// TwinCAT 3 PLC project GFT_drv_demo
// ProgramVersion: 3.1.4024.12
// libraries:
//   Tc2_EtherCAT, * (Beckhoff Automation GmbH)
//   Tc2_Standard, * (Beckhoff Automation GmbH)
//   Tc2_SUPS, * (Beckhoff Automation GmbH)
//   Tc2_System, * (Beckhoff Automation GmbH)
//   Tc2_Utilities, * (Beckhoff Automation GmbH)
//   Tc3_Module, * (Beckhoff Automation GmbH)
//   VisuDialogs, * (System)
//   VisuSymbols,3.5.10.0,System
// project tree:
//   DUTs/ CSdo_State.TcDUT, Ds402_CW.TcDUT, Ds402_Params.TcDUT, Ds402_States.TcDUT, Ds402_SW.TcDUT, E_ModesOfOperation.TcDUT, E_Notes.TcDUT, E_PosTest.TcDUT, E_SquareWave.TcDUT, E_Tests.TcDUT, Mus_Sounds.TcDUT
//   Function Blocks/ FB_Sequence.TcPOU, Profil_CSP.TcPOU
//   / GlobalTextList.TcGTLO, PlcTask.TcTTO, PlcTask_10ms.TcTTO, Visualization Manager.TcVMO (not stored)
//   GVLs/ Ds402.TcGVL, FurElise.TcGVL, GVL_IO.TcGVL, ServoCtrl.TcGVL
//   Image/ ImagePool.TcIPO (not stored)
//   POUs/ FB_PosTest.TcPOU, FB_SineSeq.TcPOU, FB_SquareWave.TcPOU, FB_GetMasterTs.TcPOU, InitSDO.TcPOU, InitSDO_w.TcPOU, MAIN.TcPOU, Main_10ms.TcPOU, MotorOn.TcPOU, OpenExplorer.TcPOU, Prg_GetClock.TcPOU, Prg_logEvents.TcPOU, Prg_WritePersistentVars.TcPOU, processStatusWord.TcPOU, Sequence.TcPOU, TestTorqueProfile.TcPOU
//   RunLog/ F_RunLogSnValid.TcPOU, FB_RunLogger.TcPOU, GVL_RunLog.TcGVL
//   Screen/ Alarm.TcVIS, Control_Panel.TcVIS, Graph.TcVIS, Overview.TcVIS, Overview_ATP.TcVIS, Servo.TcVIS, Settings.TcVIS, Password.TcVIS
//   VISUs/ Visualization.TcVIS
// real-time tasks:
//   TASK PlcTask: cycle T#1ms, priority 8, ADS port 350
//   TASK VISU_TASK: cycle T#200000us, priority 30, ADS port 351
//   TASK PlcTask_10ms: cycle T#10ms, priority 21, ADS port 352
// I/O:
//   DEVICE Device 3 (EtherCAT) (disabled), AmsNetId 5.53.59.176.4.1
//     Term 2 (EK1100) [EK1100 EtherCAT Coupler (2A E-Bus)]
//       Term 3 (EL1859) [EL1859 8Ch. Dig. Input 24V, 3ms, 8Ch. Dig. Output 24V, 0.5A]
//       Term 4 (EL2798) [EL2798 8Ch. Dig. Output 24V AC/DC, 2A, potential-free]
//       Term 5 (EL9011) [EL9011 End Terminal]
//     Box 1 (DOL Drive) [DOL Drive]
// variable links:
//   GFT-drv-demo/GFT-drv-demo Instance <-> Device 3 (EtherCAT)/Box 1 (DOL Drive)
//     PlcTask Inputs/ServoCtrl.ActualCurrent <-> TxPdo-Position-Velocity-Torque Mapping/Torque actual value
//     PlcTask Inputs/ServoCtrl.Position <-> TxPdo-Velocity Mapping/Position actual value
//     PlcTask Inputs/ServoCtrl.StatusWord <-> TxPdo-Velocity Mapping/Statusword
//     PlcTask Outputs/ServoCtrl.ControlWord <-> RxPdo-Position-Velocity-Torque Mapping/Controlword
//     PlcTask Outputs/ServoCtrl.Max_torque0x6072 <-> RxPdo-Position-Velocity-Torque Mapping/Maximal torque
//     PlcTask Outputs/ServoCtrl.ModeOfOperation <-> RxPdo-Position-Velocity-Torque Mapping/Modes of operation
//     PlcTask Outputs/ServoCtrl.PosTarget <-> RxPdo-Position-Velocity-Torque Mapping/Target position
//     PlcTask Outputs/ServoCtrl.TargetTorque <-> RxPdo-Position-Velocity-Torque Mapping/Target Torque
//     PlcTask Outputs/ServoCtrl.Target_velocity0x60FF <-> RxPdo-Position-Velocity-Torque Mapping/Target velocity
//   GFT-drv-demo/GFT-drv-demo Instance <-> Device 3 (EtherCAT)/Term 2 (EK1100)/Term 3 (EL1859)
//     PlcTask Inputs/GVL_IO.ixEmergancy_Stop <-> Channel 1/GVL_IO.ixEmergancy_Stop
//     PlcTask Inputs/GVL_IO.ixGripperLock_1 <-> Channel 4/GVL_IO.ixGripperLock_1
//     PlcTask Inputs/GVL_IO.ixGripperLock_2 <-> Channel 5/GVL_IO.ixGripperLock_1
//     PlcTask Inputs/GVL_IO.ixGripper_Unlock <-> Channel 3/GVL_IO.ixGripper_Unlock
//     PlcTask Inputs/GVL_IO.ixHome_Position <-> Channel 2/GVL_IO.ixHome_Position
//     PlcTask Outputs/GVL_IO.qxEPO_Active <-> Channel 9/GVL_IO.qxEPO_Active
//     PlcTask Outputs/GVL_IO.qxSTO_toDrive <-> Channel 16/GVL_IO.qxSTO_toDrive
//   GFT-drv-demo/GFT-drv-demo Instance <-> Device 3 (EtherCAT)/Term 2 (EK1100)/Term 4 (EL2798)
//     PlcTask Outputs/GVL_IO.qxActuator_1 <-> Channel 1/GVL_IO.qxActuator_1
//     PlcTask Outputs/GVL_IO.qxActuator_2 <-> Channel 2/GVL_IO.qxActuator_2
//     PlcTask Outputs/GVL_IO.qxBrakeOpen <-> Channel 3/GVL_IO.qxBrakeOpen

CONFIGURATION GFT_drv_demo
    RESOURCE PLC ON TwinCAT3
        TASK PlcTask(INTERVAL := T#1ms, PRIORITY := 8);
        TASK PlcTask_10ms(INTERVAL := T#10ms, PRIORITY := 21);
        PROGRAM MAIN WITH PlcTask : MAIN;
        PROGRAM Main_10ms WITH PlcTask_10ms : Main_10ms;
    END_RESOURCE
END_CONFIGURATION

// ---- DUTs/CSdo_State.TcDUT
TYPE CSdo_State :
STRUCT
	nIndex          : WORD;
	nSubIndex       : BYTE;
	bExecute        : BOOL := TRUE;
	bError			: BOOL;
	nErrId 			: UDINT;
	nBufLen   		: UDINT; 
	pBuf			: PVOID;	
END_STRUCT
END_TYPE

// ---- DUTs/Ds402_CW.TcDUT

TYPE Ds402_CW:
STRUCT 
	ReadyToSwitchOn : BOOL;// = bitand(sw,1);
	SwitchOn : BOOL;//= bitand(bitshift(sw,-1),1);
	OperationEnabled : BOOL;// = bitand(bitshift(sw,-2),1);
	Fault : BOOL;// = bitand(bitshift(sw,-3),1);
	VoltageEnabled : BOOL;// = bitand(bitshift(sw,-4),1);
	NoQuickStop : BOOL;// = bitand(bitshift(sw,-5),1);
	SwitchOnDisabled : BOOL;// = bitand(bitshift(sw,-6),1);
	Warning : BOOL;// = bitand(bitshift(sw,-7),1);
	ManufacturerSpecific8 : BOOL;// = bitand(bitshift(sw,-8),1);
	Remote : BOOL;// = bitand(bitshift(sw,-9),1);
	TargetReached : BOOL;// = bitand(bitshift(sw,-10),1);
	InternalLimitActive : BOOL;// = bitand(bitshift(sw,-11),1);
	OperationModeSpecific12to13 : INT;// = bitand(bitshift(sw,-12),3);
	ManufacturerSpecific14to15 : INT;// = bitand(bitshift(sw,-14),3);
END_STRUCT
END_TYPE

// ---- DUTs/Ds402_Params.TcDUT
TYPE Ds402_Params :
STRUCT
	Motor_rated_torque0x6076 : UDINT;
	Interpolation_time_period0x60C2_1_period : USINT;
	Interpolation_time_period0x60C2_2_period : SINT;
	vendorId_0x1081_1 : UDINT;
	Postion_window0x6067 : UDINT;
	Position_window_time0x6068 :  UINT;
	Abort_connection_option_code_0x6007 :  UINT;
	Torque_slope0x6087 :    UDINT;
END_STRUCT
END_TYPE

// ---- DUTs/Ds402_States.TcDUT
{attribute 'qualified_only'}
{attribute 'strict'}
(*
TYPE Ds402_States :
(
	FSM_Ilegal := -2 ;
	FSM_NotReadyToSwitchOn := -1 ; 
	FSM_SwitchOnDisabled  := 0 ;
	FSM_ReadyToSwitchOn := 1;
	FSM_SwitchedOn := 2;
	FSM_OperationEnabled := 3 ;
	FSM_QuickStopActive := 4 ;
	FSM_FaultReactionActive := 5;
	FSM_Fault := 6 ; 
	FSM_Temporary_Fault := 7; 
);
END_TYPE
*)
;

// ---- DUTs/Ds402_SW.TcDUT
TYPE Ds402_SW :
STRUCT
	ReadyToSwitchOn : BOOL;// = bitand(sw,1);
	SwitchOn : BOOL;//= bitand(bitshift(sw,-1),1);
	OperationEnabled : BOOL;// = bitand(bitshift(sw,-2),1);
	Fault : BOOL;// = bitand(bitshift(sw,-3),1);
	VoltageEnabled : BOOL;// = bitand(bitshift(sw,-4),1);
	NoQuickStop : BOOL;// = bitand(bitshift(sw,-5),1);
	SwitchOnDisabled : BOOL;// = bitand(bitshift(sw,-6),1);
	Warning : BOOL;// = bitand(bitshift(sw,-7),1);
	ManufacturerSpecific8 : BOOL;// = bitand(bitshift(sw,-8),1);
	Remote : BOOL;// = bitand(bitshift(sw,-9),1);
	TargetReached : BOOL;// = bitand(bitshift(sw,-10),1);
	InternalLimitActive : BOOL;// = bitand(bitshift(sw,-11),1);
	OperationModeSpecific12to13 : INT;// = bitand(bitshift(sw,-12),3);
	ManufacturerSpecific14to15 : INT;// = bitand(bitshift(sw,-14),3);

	SetPointAck:   BOOL ;// bitand(bitshift(sw,-12),1);
	FollowingError:BOOL ; // bitand(bitshift(sw,-13),1);

END_STRUCT
END_TYPE

// ---- DUTs/E_ModesOfOperation.TcDUT
{attribute 'qualified_only'}
{attribute 'strict'}
TYPE E_ModesOfOperation :
(
	ED_MO_NoModeChange := 0 , 
	ED_MO_Profile_position_mode := 1 , 
	ED_MO_Profile_velocity_mode := 3 , 
	ED_MO_Torque_profile_mode := 4, 
	ED_MO_Inertial_profile_mode := 5, 
	ED_MO_Homing_mode := 6, 
	ED_MO_Interpolated_position_mode := 7, 
	ED_MO_Cyclic_sync_position_mode := 8, 
	ED_MO_Cyclic_sync_velocity_mode := 9, 
	ED_MO_Cyclic_sync_torque_mode := 10,
	ED_MO_Profile_only_velocity_mode := 11,
	ED_MO_Profile_test_wave_mode := 12,
	ED_MO_User_Prj_spec_mode := 13
);
END_TYPE

// ---- DUTs/E_Notes.TcDUT
{attribute 'qualified_only'}
{attribute 'strict'}
TYPE E_Notes :
(
STOP     := 0,
PAUSE    := 1,
NOTE_B0  := 31  ,
NOTE_C1  := 33  ,
NOTE_CS1 := 35  ,
NOTE_D1  := 37  ,
NOTE_DS1 := 39  ,
NOTE_E1  := 41  ,
NOTE_F1  := 44  ,
NOTE_FS1 := 46  ,
NOTE_G1  := 49  ,
NOTE_GS1 := 52  ,
NOTE_A1  := 55  ,
NOTE_AS1 := 58  ,
NOTE_B1  := 62  ,
NOTE_C2  := 65  ,
NOTE_CS2 := 69  ,
NOTE_D2  := 73  ,
NOTE_DS2 := 78  ,
NOTE_E2  := 82  ,
NOTE_F2  := 87  ,
NOTE_FS2 := 93  ,
NOTE_G2  := 98  ,
NOTE_GS2 := 104 ,
NOTE_A2  := 110 ,
NOTE_AS2 := 117 ,
NOTE_B2  := 123 ,
NOTE_C3  := 131 ,
NOTE_CS3 := 139 ,
NOTE_D3  := 147 ,
NOTE_DS3 := 156 ,
NOTE_E3  := 165 ,
NOTE_F3  := 175 ,
NOTE_FS3 := 185 ,
NOTE_G3  := 196 ,
NOTE_GS3 := 208 ,
NOTE_A3  := 220 ,
NOTE_AS3 := 233 ,
NOTE_B3  := 247 ,
NOTE_C4  := 262 ,
NOTE_CS4 := 277 ,
NOTE_D4  := 294 ,
NOTE_DS4 := 311 ,
NOTE_E4 := 330 ,
NOTE_F4  := 349 ,
NOTE_FS4 := 370 ,
NOTE_G4  := 392 ,
NOTE_GS4 := 415 ,
NOTE_A4  := 440 ,
NOTE_AS4 := 466 ,
NOTE_B4  := 494 ,
NOTE_C5  := 523 ,
NOTE_CS5 := 554 ,
NOTE_D5  := 587 ,
NOTE_DS5 := 622 ,
NOTE_E5  := 659 ,
NOTE_F5  := 698 ,
NOTE_FS5 := 740 ,
NOTE_G5  := 784 ,
NOTE_GS5 := 831 ,
NOTE_A5  := 880 ,
NOTE_AS5 := 932 ,
NOTE_B5  := 988 ,
NOTE_C6  := 1047,
NOTE_CS6 := 1109,
NOTE_D6  := 1175,
NOTE_DS6 := 1245,
NOTE_E6  := 1319,
NOTE_F6  := 1397,
NOTE_FS6 := 1480,
NOTE_G6  := 1568,
NOTE_GS6 := 1661,
NOTE_A6  := 1760,
NOTE_AS6 := 1865,
NOTE_B6  := 1976,
NOTE_C7  := 2093,
NOTE_CS7 := 2217,
NOTE_D7  := 2349,
NOTE_DS7 := 2489,
NOTE_E7  := 2637,
NOTE_F7  := 2794,
NOTE_FS7 := 2960,
NOTE_G7  := 3136,
NOTE_GS7 := 3322,
NOTE_A7  := 3520,
NOTE_AS7 := 3729,
NOTE_B7  := 3951,
NOTE_C8  := 4186,
NOTE_CS8 := 4435,
NOTE_D8  := 4699,
NOTE_DS8 := 4978
);
	
END_TYPE

// ---- DUTs/E_PosTest.TcDUT
{attribute 'qualified_only'}
{attribute 'strict'}
TYPE E_PosTest :
(
	Idle_start :=0,
	GoToNextState_levelHi := 1,
	GoToNextState_levelLo := 2,
	MovingTo_levelHi :=3,
	MovingTo_levelLo :=4,
	Idle_init :=5
);
END_TYPE

// ---- DUTs/E_SquareWave.TcDUT
{attribute 'qualified_only'}
{attribute 'strict'}
TYPE E_SquareWave :
(
	GoToNextState_levelHi := 1,
	GoToNextState_levelLo :=2,
	GoToNextState_Off :=3
);
END_TYPE

// ---- DUTs/E_Tests.TcDUT
{attribute 'qualified_only'}
{attribute 'strict'}
TYPE E_Tests :
(
	E_Current_SquareWaveTest := 1,
	E_Current_SinWaveTest := 2,
	E_Position_Ptp := 3,
	E_Position_Csp := 4,
	E_Velocity_Csv :=5
);
END_TYPE

// ---- DUTs/Mus_Sounds.TcDUT
TYPE Mus_Sounds :
STRUCT
	note : E_Notes;
	tempo: INT;
END_STRUCT
END_TYPE

// ---- GVLs/Ds402.TcGVL
{attribute 'qualified_only'}


VAR_GLOBAL
	StatusWord_Bits :  Ds402_SW;
	DirUp : BOOL;
	ProfParams : Ds402_Params;

END_VAR

// ---- GVLs/FurElise.TcGVL
{attribute 'qualified_only'}
VAR_GLOBAL CONSTANT
	FurElise : ARRAY [0..100] OF  Mus_Sounds :=[
 	(note := E_Notes.NOTE_E5,              tempo:= 9),
                (note := E_Notes.NOTE_DS5,  tempo:=    9),
                (note := E_Notes.NOTE_E5,    tempo:=   9),
                (note := E_Notes.NOTE_DS5,   tempo:=   9),
                (note := E_Notes.NOTE_E5,    tempo:=   9),
                (note := E_Notes.NOTE_B4,    tempo:=   9),
                (note := E_Notes.NOTE_D5,    tempo:=   9),
                (note := E_Notes.NOTE_C5,    tempo:=   9),
                (note := E_Notes.NOTE_A4,    tempo:=   3),
                (note := E_Notes.NOTE_C4,    tempo:=   9),
                (note := E_Notes.NOTE_E4,    tempo:=   9),
                (note := E_Notes.NOTE_A4,    tempo:=   9),
                (note := E_Notes.NOTE_B4,     tempo:=  3),
                (note := E_Notes.NOTE_E4,    tempo:=   9),
                (note := E_Notes.NOTE_GS4,    tempo:=  9),
                (note := E_Notes.NOTE_B4,    tempo:=          9),
                (note := E_Notes.NOTE_C5,    tempo:=   3),
                (note := E_Notes.NOTE_E4,    tempo:=   9),
                (note := E_Notes.NOTE_E5,    tempo:=   9),
                (note := E_Notes.NOTE_DS5,   tempo:=   9),
                (note := E_Notes.NOTE_E5,    tempo:=   9),
                (note := E_Notes.NOTE_DS5,   tempo:=   9),
                (note := E_Notes.NOTE_E5,    tempo:=   9),
                (note := E_Notes.NOTE_B4,    tempo:=   9),
                (note := E_Notes.NOTE_D5,   tempo:=    9),
                (note := E_Notes.NOTE_C5,   tempo:=    9),
                (note := E_Notes.NOTE_A4,    tempo:=   3),
                (note := E_Notes.NOTE_C4,    tempo:=   9),
                (note := E_Notes.NOTE_E4,    tempo:=   9),
                (note := E_Notes.NOTE_A4,    tempo:=   9),
                (note := E_Notes.NOTE_B4,    tempo:=   3),
                (note := E_Notes.NOTE_E4,    tempo:=          9),
                (note := E_Notes.NOTE_C5,    tempo:=   9),
                (note := E_Notes.NOTE_B4,   tempo:=    9),
                (note := E_Notes.NOTE_A4,    tempo:=   3),
                (note := E_Notes.NOTE_B4,    tempo:=   9),
                (note := E_Notes.NOTE_C5,    tempo:=   9),
                (note := E_Notes.NOTE_D5,    tempo:=   9),
                (note := E_Notes.NOTE_E5,    tempo:=   3),
                (note := E_Notes.NOTE_G4,    tempo:=   9),
                (note := E_Notes.NOTE_F5,    tempo:=   9),
                (note := E_Notes.NOTE_E5,    tempo:=   9),
                (note := E_Notes.NOTE_D5,     tempo:=  3),
                (note := E_Notes.NOTE_F4,     tempo:=  9),
                (note := E_Notes.NOTE_E5,    tempo:=   9),
                (note := E_Notes.NOTE_D5,    tempo:=   9),
                (note := E_Notes.NOTE_C5,    tempo:=   3),
                (note := E_Notes.NOTE_E4,    tempo:=          9),
                (note := E_Notes.NOTE_D5,   tempo:=    9),
                (note := E_Notes.NOTE_C5,    tempo:=   9),
                (note := E_Notes.NOTE_B4,    tempo:=   9),
                (note := E_Notes.NOTE_E4,    tempo:=   9),
                (note := E_Notes.NOTE_E5,   tempo:=    9),
                (note := E_Notes.NOTE_E4,    tempo:=   9),
                (note := E_Notes.NOTE_E5,    tempo:=   9),
                (note := E_Notes.NOTE_E4,    tempo:=   9),
                (note := E_Notes.NOTE_E5,    tempo:=   9),
                (note := E_Notes.NOTE_E4,     tempo:=  9),
                (note := E_Notes.NOTE_E5,    tempo:=   9),
                (note := E_Notes.NOTE_DS4,    tempo:=  9),
                (note := E_Notes.NOTE_E5,    tempo:=   9),
                (note := E_Notes.NOTE_D4,     tempo:=  9),
                (note := E_Notes.NOTE_E5,     tempo:=  9),
                (note := E_Notes.NOTE_DS4,   tempo:=        9),
                (note := E_Notes.NOTE_E5,    tempo:=   9),
                (note := E_Notes.NOTE_B4,    tempo:=   9),
                (note := E_Notes.NOTE_D5,    tempo:=   9),
                (note := E_Notes.NOTE_C5,    tempo:=   9),
                (note := E_Notes.NOTE_A4,     tempo:=  3),
                (note := E_Notes.NOTE_C4,     tempo:=  9),
                (note := E_Notes.NOTE_E4,    tempo:=   9),
                (note := E_Notes.NOTE_A4,    tempo:=   9),
                (note := E_Notes.NOTE_B4,    tempo:=   3),
                (note := E_Notes.NOTE_E4,    tempo:=   9),
                (note := E_Notes.NOTE_GS4,   tempo:=   9),
                (note := E_Notes.NOTE_B4,     tempo:=  9),
                (note := E_Notes.NOTE_C5,     tempo:=  3),
                (note := E_Notes.NOTE_E4,     tempo:=  9),
                (note := E_Notes.NOTE_E5,     tempo:=  9),
                (note := E_Notes.NOTE_DS5,    tempo:=       9),
                (note := E_Notes.NOTE_E5,    tempo:=   9),
                (note := E_Notes.NOTE_DS5,    tempo:=  9),
                (note := E_Notes.NOTE_E5,     tempo:=  9),
                (note := E_Notes.NOTE_B4,     tempo:=  9),
                (note := E_Notes.NOTE_D5,     tempo:=  9),
                (note := E_Notes.NOTE_C5,     tempo:=  9),
                (note := E_Notes.NOTE_A4,    tempo:=   3),
                (note := E_Notes.NOTE_C4,    tempo:=   9),
                (note := E_Notes.NOTE_E4,    tempo:=   9),
                (note := E_Notes.NOTE_A4,    tempo:=   9),
                (note := E_Notes.NOTE_B4,    tempo:=   3),
                (note := E_Notes.NOTE_E4,    tempo:=   8),
                (note := E_Notes.NOTE_C5,    tempo:=   8),
                (note := E_Notes.NOTE_B4,    tempo:=   8),
                (note := E_Notes.NOTE_A4,    tempo:=   1),
                (note := E_Notes.STOP,       tempo:=   9)
];

END_VAR

// ---- GVLs/GVL_IO.TcGVL
{attribute 'qualified_only'}
VAR_GLOBAL
	
	// Digital Input
	ixGripper_Up AT%I*:BOOL;
	ixEncoder AT%I*:BOOL;
	ixHome_Position AT%I*:BOOL;
	ixEmergancy_Stop AT%I*:BOOL;
	ixGripperLock_1 AT%I*:BOOL;
	ixGripperLock_2 AT%I*:BOOL;
	ixGripper_Unlock AT%I*:BOOL;
	ixGripperLock_A AT%I*:BOOL;
	ixGripperLock_B AT%I*:BOOL;
	
	
	//MOtor input
	Velosity_PV AT%I*:DINT;
	
	// Digital Output
	qxStart_Motor AT%Q*:BOOL;
	qxOpen_Gripper AT%Q*:BOOL;
	qxGripper_UP AT%Q*:BOOL;
	qxSTO_toDrive AT%Q*:BOOL;
	qxEPO_Active AT%Q*:BOOL;
	qxClose_Gripper AT%Q*:BOOL;
	qxBrakeOpen AT%Q*:BOOL;
	qxActuator_1 AT%Q*:BOOL; 	// Direction : 0 - close; 1 - open
	qxActuator_2 AT%Q*:BOOL;	// command Move 
	
	// Global
	Reset, Homing, Motor_UP, Motor_DN, Gripper_Open_cmd, Gripper_Close_cmd, Jog_UP, Jog_DN , Zeroing_cmd: BOOL;
	Position_PV, Position_SP, Motor_I , Position_PV_HMI, Position_PV_Diff: DINT;
	 
	Motor_I_PV, Motor_I_MAX, Motor_I_AVR : REAL;
	Motor_I_mem : ARRAY [0..500] OF REAL;
	Position_PV_mem : ARRAY [0..500] OF DINT;
	
	
	Enable, Emergancy_OK, Motor_UP_cmd, Motor_DN_cmd, Homing_OK, Homing_cmd , TwoSensorLock:BOOL;
	Step, Gripper_step:INT;
	Always_ON, Always_OFF, FirstScan :BOOL;
	GO_TO_cmd, Motion_in_Progress, Ready_for_start, Start, Stop, Run_Cycle, Enable_motor_cmd:BOOL;
	tonHomingError_IN, tonHomingStepDelay_IN : BOOL;
	tonHomingStepDelay_SP : TIME;
	
	 
	
	
	Position_UP_SP_LL, Position_UP_SP_HL, Position_DN_SP_LL, Position_DN_SP_HL : DINT;
	Cycle_PV: UDINT;
	UP_pause_in:BOOL;
	Error, Gripper_Open_Error, Gripper_Close_Error , Emergancy_Error, SensorLock_Error, Homing_Error, Motor_Error: BOOL;
	Position_sp_test : DINT;
	pp, pv :REAL;
	Speed_SP_mem, Accseleration_SP_mem : REAL;
	tonUserDelay_IN, tonUserDelay_Q, tonMotionError_IN, tonMotionError_Q : BOOL;
	tonLogTimer_IN , tonLogTimer_Q : BOOL;
	Password : INT := 9118 ;
	Password_IN : INT;
	
	Calc_log_cmd , OpenExplorer_cmd, New_CSV_cmd : BOOL;
	Lod_appendLine_cmd, Log_CloseFile_cmd : BOOL;
	Log_nMode : DWORD;
	Log_Data, Motor_UP_slow_cmd, Motor_DN_slow_cmd , Slow_cycle_cmd , ATP_start_cmd: BOOL;	
	test_Gripper_open_OK, test_Gripper_close_OK, test_motor_sldown_ok, test_motor_slUP_ok, test_Insert_OK, test_slowCycle_OK : BOOL;
		
	
	
	
END_VAR

VAR_GLOBAL PERSISTENT
	vcc_SP : REAL ; //:= 4000000;
	acc_SP: REAL ; //:= 80000000;
    Position_UP_SP, Position_DN_SP : DINT;
	Position_UP_A_SP, Position_DN_A_SP : DINT; // position  Accseleration Change
	Speed_SP, Accseleration_SP , Accseleration_A_SP: REAL;
	Speed_SP_slow, Accseleration_SP_slow : REAL;
	Cycle_SP : UDINT;
	Motor_Limit_UP, Motor_Limit_DN :DINT; 
	
	
	
	
END_VAR

// ---- GVLs/ServoCtrl.TcGVL
{attribute 'qualified_only'}
VAR_GLOBAL
	TargetTorque AT %Q*: INT;
	TorqueProfState: REAL;
	PosTarget  AT %Q*: DINT;
	Position  AT %I*: DINT ;
	ControlWord AT %Q*: UINT;
	StatusWord AT %I*:  INT ;
	ActualCurrent AT %I*:  DINT ;
	ModeOfOperation AT %Q*: SINT;
	PosSensor1 AT %I*:  DINT ;
	PosSensor2 AT %I*:  DINT ;
	Max_torque0x6072 AT %Q*: UINT;
	Target_velocity0x60FF AT %Q*: DINT;
END_VAR

// ---- RunLog/GVL_RunLog.TcGVL
// Run log module: what the HMI shows and enters. Format: report-tool/docs/log-format.md
{attribute 'qualified_only'}
VAR_GLOBAL
	SN			: STRING(32);	// part serial number, entered on Overview_ATP before START
	SN_valid	: BOOL;			// 1..32 characters of A-Z a-z 0-9 -; ATP START needs it
	State		: STRING(40);	// what the logger is doing now
	LastFile	: STRING(255);	// last finished run log
	LastError	: STRING(255);	// last problem; a run without a valid SN is not logged
	ErrorCount	: UDINT;
END_VAR

// ---- POUs/MAIN.TcPOU
PROGRAM MAIN
VAR

testType : E_Tests :=E_Tests.E_Position_Csp;// E_Tests.E_Velocity_Csv;//E_Tests.E_Position_Csp;//E_Tests.E_Current_SinWaveTest;//E_Tests.E_Position_Ptp;

ApplyPosTargetNow : BOOL := FALSE;
//ModeOfOperation : SINT := TO_SINT(E_ModesOfOperation.ED_MO_Cyclic_sync_torque_mode);// ED_MO_Cyclic_sync_torque_mode
bInitDone : BOOL :=FALSE;
bInitDone_w : BOOL :=FALSE;//finished SDO download to slave

valueA : UDINT;
sNetId     : T_AmsNetId := '5.53.59.176.4.1'; // '5.53.59.176.1.1';
nSlaveAddr : UINT := 1001;
//fbSdoRead  : FB_EcCoESdoRead;
//sdo1_err : BOOL;
//sdo1_nErrId : UDINT;
//sdo1_value  :  UDINT;
//sdo1_value_size  :  UDINT := SIZEOF(sdo1_value);

TorCmd_ds402  :  INT :=0;
TorCmdMax_Ds402 :  UINT :=0;
TorCmdA : REAL := 4;
TorCmdMaxA : REAL := 17;
FreqScale : REAL := 0.25;
ProfParams: Ds402_Params;// uploaded from slave
ProfParams_w: Ds402_Params;// to download to slave
// State machine
fbSquareWave		: FB_SquareWave;
fbMusic : FB_SineSeq;
fbInitSDO_w : InitSDO_w;// write SDO to slave
fbInitSDO : InitSDO;// read SDO from slave
fbPosTest : FB_PosTest; // position profiler test

	bInit_Sdo_States : BOOL :=TRUE;
//	indSdo :   USINT :=0;
//	Sdo_States : ARRAY [0..10] OF CSdo_State ;
	TaskTotalTime : UDINT;
	fbGetMasterTs : FB_GetMasterTs;
	cpu_info : ARRAY [0..10] of ST_CpuCoreInfo;
	FB_Sequence_DB: FB_Sequence;
	Profile_CSP_DB: Profil_CSP;
	
	
	
	
END_VAR


TaskTotalTime := F_GetTaskTotalTime(0);// x100ns 
fbGetMasterTs();
F_GetCpuCoreInfo(0,ADR(cpu_info[0]));
F_GetCpuCoreInfo(0,ADR(cpu_info[1]));
 
(*
IF bInit_Sdo_States AND fbGetMasterTs.MasterTsUsec> 0 THEN
	fbInitSDO(sNetId:=sNetId,nSlaveAddr:=nSlaveAddr);
	fbInitSDO.Init();

	CASE fbGetMasterTs.MasterTsUsec OF
	100:
		ProfParams_w.Interpolation_time_period0x60C2_1_period := 10;
		ProfParams_w.Interpolation_time_period0x60C2_2_period := -5;
	200:
		ProfParams_w.Interpolation_time_period0x60C2_1_period := 20;
		ProfParams_w.Interpolation_time_period0x60C2_2_period := -5;
		
	250:
		ProfParams_w.Interpolation_time_period0x60C2_1_period := 25;
		ProfParams_w.Interpolation_time_period0x60C2_2_period := -5;
	
	500:
		ProfParams_w.Interpolation_time_period0x60C2_1_period := 5;
		ProfParams_w.Interpolation_time_period0x60C2_2_period := -4;
	1000:
		ProfParams_w.Interpolation_time_period0x60C2_1_period := 1;
		ProfParams_w.Interpolation_time_period0x60C2_2_period := -3;
	END_CASE
	ProfParams_w.Postion_window0x6067 := 200;
	ProfParams_w.Position_window_time0x6068 := 1000;
	
	ProfParams_w.Abort_connection_option_code_0x6007 := 16#0002;
	
	fbInitSDO_w(sNetId:=sNetId,nSlaveAddr:=nSlaveAddr,ProfParams:=ProfParams_w);
	fbInitSDO_w.Init();
	//FreqScale := 0.25 * 1000.0 / INT_TO_REAL(fbGetMasterTs.MasterTsUsec)   ;
	bInit_Sdo_States:= FALSE;
END_IF

IF NOT bInit_Sdo_States THEN
	fbInitSDO_w.writeSDO();
	bInitDone_w := fbInitSDO_w.bInitDone;
	IF bInitDone_w THEN
	fbInitSDO.readSDO();
	bInitDone := fbInitSDO.bInitDone;
	END_IF
END_IF
*)
bInitDone:= TRUE;
//TestTorqueProfile();
IF bInitDone THEN
	ProfParams:= fbInitSDO.ProfParams;
	
	//IF ProfParams.Motor_rated_torque0x6076 > 0 THEN
	//	TorCmd_ds402  := TRUNC_INT( TorCmdA * 1E6 / UDINT_TO_REAL(ProfParams.Motor_rated_torque0x6076));// TC*10e6/0x6076
	//	TorCmdMax_Ds402:=INT_TO_UINT( TRUNC_INT( TorCmdMaxA * 1E6 / UDINT_TO_REAL(ProfParams.Motor_rated_torque0x6076)));// TC*10e6/0x6076
	//ELSE 
	//	TorCmd_ds402  :=0;TorCmdMax_Ds402:=0;
	//END_IF
	TorCmdMax_Ds402:= 65535;//62000;
	
	// E_Current_SquareWaveTest->E_Current_SinWaveTest->E_Position_Ptp
	CASE testType OF
		E_Tests.E_Current_SquareWaveTest:
			fbSquareWave(RefLevelHi:= TorCmd_ds402,RefLevelLo:= -TorCmd_ds402);
			fbSquareWave.Execute(bCyclicMode:=FALSE);
			IF fbSquareWave.nCycles > 20 THEN
				fbSquareWave.Restart();
				testType := E_Tests.E_Current_SinWaveTest;
			END_IF
		E_Tests.E_Current_SinWaveTest:
			fbMusic(Motor_rated_torque0x6076:=ProfParams.Motor_rated_torque0x6076,
			AmpMax := TorCmdMaxA,FreqScale:= FreqScale);
			fbMusic.Execute(Mode_of_operation:= E_ModesOfOperation.ED_MO_Cyclic_sync_torque_mode);
			IF fbMusic.nCycles > 0 THEN
				fbMusic.Restart();
				testType := E_Tests.E_Position_Ptp;

			END_IF

		E_Tests.E_Position_Ptp:
			fbPosTest(PosTargetL:=90000000,PosTargetR:=1000000);
			fbPosTest.Execute();
			ApplyPosTargetNow := fbPosTest.ApplyPosTargetNow;
			IF fbPosTest.nCycles > 5 THEN
			//	fbPosTest.Restart();
			//	testType := E_Tests.E_Position_Csp;
			END_IF
		E_Tests.E_Position_Csp:
			
			fbMusic(Motor_rated_torque0x6076:=ProfParams.Motor_rated_torque0x6076,
			AmpMax := TorCmdMaxA,FreqScale:= FreqScale*0.75,
			PosOffset:=3000,PosAmp:= 100000);
			fbMusic.Execute(Mode_of_operation:= E_ModesOfOperation.ED_MO_Cyclic_sync_position_mode);
			
			IF fbMusic.nCycles > 0 THEN
				fbMusic.Restart();
			//	testType := E_Tests.E_Current_SquareWaveTest;
			END_IF
		E_Tests.E_Velocity_Csv:
			
			fbMusic(Motor_rated_torque0x6076:=ProfParams.Motor_rated_torque0x6076,
			AmpMax := TorCmdMaxA,FreqScale:= FreqScale*0.75,
			PosOffset:=3000,PosAmp:= 30000);
			fbMusic.Execute(Mode_of_operation:= E_ModesOfOperation.ED_MO_Cyclic_sync_velocity_mode);
			
			IF fbMusic.nCycles > 0 THEN
				fbMusic.Restart();
			//	testType := E_Tests.E_Current_SquareWaveTest;
			END_IF
	

	END_CASE
	

	ServoCtrl.Max_torque0x6072 := TorCmdMax_Ds402;
	
	//ApplyPosTargetNow := FALSE;
	//IF ServoCtrl.Position > 32000 THEN
	//	ServoCtrl.PosTarget := 0;
	//	ApplyPosTargetNow := TRUE;
	//END_IF
	//
	//IF ServoCtrl.Position < 100 THEN
	//	ServoCtrl.PosTarget := 32100;
	//	ApplyPosTargetNow := TRUE;
	//END_IF
	//
	//ServoCtrl.PosTarget := ServoCtrl.PosTarget +1;
	Ds402.StatusWord_Bits := processStatusWord(ServoCtrl.StatusWord);
	ServoCtrl.ControlWord := MotorOn(Ds402.StatusWord_Bits,ApplyPosTargetNow);

END_IF


// Emergancy RED LED from Door
IF NOT gvl_io.ixEmergancy_Stop
	THEN
	gvl_io.qxEPO_Active := TRUE;
	ELSE
		gvl_io.qxEPO_Active := FALSE;
END_IF



FB_Sequence_DB();
Prg_WritePersistentVars();
//Sequence();

//Prg_logEvents();
Profile_CSP_DB(
	p_in:= DINT_TO_REAL(gvl_io.Position_sp_test), 
	pold:= gvl_io.pp, 
	vold:= gvl_io.pv, 
	vcc:= gvl_io.vcc_SP, 
	acc:= gvl_IO.acc_SP, 
	Ts:= 0.001, 
	pp=> gvl_io.pp, 
	pv=> gvl_io.pv);

END_PROGRAM

// ---- POUs/FB_SquareWave.TcPOU
FUNCTION_BLOCK FB_SquareWave
VAR_INPUT
	RefLevelHi : INT := 0;
	RefLevelLo : INT := 0;
	bGoToOffState : BOOL := FALSE;
END_VAR
VAR_OUTPUT
	OutRef : INT :=0;
		nCycles : DINT := 0;

END_VAR
VAR
	eStateMachine		: E_SquareWave :=E_SquareWave.GoToNextState_levelHi;
	nCounterState1		: INT;
	nCounterState2		: INT;
//	nCounterState3		: INT;
	fbTimer				: TON;
	tGoToNextState1		: TIME := T#0.5S;
	tGoToNextState2		: TIME := T#0.8S;
	fbTrigger			: R_TRIG;
//	bGoToNextState		: BOOL;

END_VAR

METHOD Execute : BOOL
VAR_INPUT
	bCyclicMode : BOOL := FALSE; 
END_VAR
CASE eStateMachine OF
	
E_SquareWave.GoToNextState_Off:
	OutRef:=0;
	
E_SquareWave.GoToNextState_levelHi:
	// Increase counter to show that state 1 is active
	nCounterState1 := nCounterState1 + 1;
	OutRef := RefLevelHi;
	// Call timer FB with the desired time parameter
	// In the first execution of this state, "fbTimer" is activated by a rising edge at the execute input "IN".
	// PLEASE REMARK: Afterwards, the FB has to be called in each following cycle until the time has run off.
	// When the time has run off, the output Q becomes TRUE and the timer FB is called with an input reset.
	// Then, the FB does not have to be called anymore - until it should be activated with a rising edge at the execute input again.
	fbTimer(IN := TRUE,
			PT := tGoToNextState1);
			
	// Check if the time has run off
	IF fbTimer.Q THEN
		fbTimer(IN := FALSE);											// Reset timer FB by resetting the execute input "IN"
		eStateMachine := E_SquareWave.GoToNextState_levelLo;	// Switch to next state
	nCycles:=nCycles+1;
	END_IF

E_SquareWave.GoToNextState_levelLo:
	// Increase counter to show that state 1 is active
	nCounterState2 := nCounterState2 + 1;
	OutRef := RefLevelLo;

	fbTimer(IN := TRUE,
			PT := tGoToNextState1);
			
	// Check if the time has run off
	IF fbTimer.Q THEN
		fbTimer(IN := FALSE);											// Reset timer FB by resetting the execute input "IN"
		eStateMachine := E_SquareWave.GoToNextState_levelHi;	// Switch to next state
	END_IF
	
	
END_CASE

// Call trigger FB to detect a rising edge of the connected variable/condition
// => User interaction necessary: To switch to the next state, write the variable "bGoToNextState" to TRUE
fbTrigger(CLK := bGoToOffState);

// Check if the trigger detected a rising edge
IF fbTrigger.Q THEN
//	bGoToNextState	:= FALSE;										// Reset control variable
	eStateMachine	:= E_SquareWave.GoToNextState_Off;		// Switch to next state
END_IF
ServoCtrl.TargetTorque := OutRef;
IF bCyclicMode THEN
	ServoCtrl.ModeOfOperation := TO_SINT(E_ModesOfOperation.ED_MO_Cyclic_sync_torque_mode);
ELSE
	ServoCtrl.ModeOfOperation := TO_SINT(E_ModesOfOperation.ED_MO_Torque_profile_mode);
END_IF
END_METHOD

METHOD Restart : BOOL
VAR_INPUT
END_VAR
		nCycles   := 0;
		eStateMachine :=E_SquareWave.GoToNextState_levelHi;
END_METHOD

END_FUNCTION_BLOCK

// ---- POUs/FB_SineSeq.TcPOU
FUNCTION_BLOCK FB_SineSeq
VAR_INPUT
//	RefLevelHi : INT := 0;
//	RefLevelLo : INT := 0;
//	bGoToOffState : BOOL := FALSE;
	Motor_rated_torque0x6076 : UDINT;
	AmpMax : REAL ;
	bSingleFreq :BOOL:=FALSE;
	SingleFreqHz : REAL:=100; 
	FreqScale : REAL :=0.25;
	PosOffset : DINT :=0;
	PosAmp 		: UDINT :=0;
	
END_VAR
VAR_OUTPUT
	OutRef : INT :=0;
	OutRefP : DINT :=0;
	
		nCycles : DINT := 0;

END_VAR
VAR
	Amp  : REAL := 0;
	FreqHz : REAL := 1;
	nFullCycles : REAL;
	Ph : real :=0;
	ind : INT :=0;
 //TorCmdMax : DINT := TRUNC( 3.0 * 1E6 / 10000);// TC*10e6/0x6076
 tTimerValue     : LTIME ;//:= T#0S;
 tTimeHr,tTimeHrPrev : UDINT;
 dTTimeHr : UDINT;
	eStateMachine		: E_SquareWave;
	nCounterState1		: INT;
	nCounterState2		: INT;
//	nCounterState3		: INT;
	fbTimer				: TON;
	tGoToNextState1		: TIME := T#2.0S;
//	tGoToNextState2		: TIME := T#0.8S;
		duration: TIME := T#1.0S;
//	fbTrigger			: R_TRIG;
//	bGoToNextState		: BOOL;

END_VAR

METHOD Execute : BOOL
VAR_INPUT
	Mode_of_operation  : E_ModesOfOperation ;
END_VAR
VAR
	TorCmd_ds402 : INT;
//	w : REAL;
	F : REAL;
//	Profile_CSP_DB: Profil_CSP;
	
	
END_VAR

//IF eStateMachine  = E_SquareWave.GoToNextState_levelHi THEN
	fbTimer(IN := TRUE,
			PT := duration);
	//eStateMachine := E_SquareWave.GoToNextState_levelLo;
//END_IF
			
	// Check if the time has run off
	IF fbTimer.Q THEN
		fbTimer(IN := FALSE);											// Reset timer FB by resetting the execute input "IN"
		//eStateMachine := E_SquareWave.GoToNextState_levelLo;	// Switch to next state
		ind	:=ind+1;
	END_IF

	

IF FurElise.FurElise[ind].note <> E_Notes.STOP AND ind < 100 THEN
	IF FurElise.FurElise[ind].note = E_Notes.pause THEN
			Amp := 0;
	ELSE
			Amp := AmpMax;
	END_IF
	F := FurElise.FurElise[ind].note;
	FreqHz := F * FreqScale;
	IF bSingleFreq THEN
		FreqHz := SingleFreqHz;
	END_IF
		
	nFullCycles := INT_TO_REAL( TRUNC_INT(FreqHz*1E-9* UDINT_TO_REAL(16#40000000)) );

	// duration = 1000 / tempo (ms)
	duration := tGoToNextState1 / FurElise.FurElise[ind].tempo;
	//ind:=ind+1;
ELSE
	ind:=0;// infinite
	nCycles := nCycles+1;
END_IF

tTimerValue := LTIME();

tTimeHrPrev := tTimeHr;
tTimeHr := LTIME_TO_UDINT(tTimerValue) MOD  16#40000000 ;
dTTimeHr :=(tTimeHr-tTimeHrPrev);// [nsec]
// for Ts = 1ms
Ph:=UDINT_TO_REAL( tTimeHr) * 6.283185307179586 *nFullCycles / UDINT_TO_REAL(16#40000000);
//for Ts=100usec: ServoCtrl.TargetTorque := TRUNC_INT( TorCmdMax * SIN(  tTimeHr * 6.28 *32.0 / 67108864.0 ));

CASE  Mode_of_operation OF
E_ModesOfOperation.ED_MO_Cyclic_sync_position_mode:
		OutRefP := TRUNC( UDINT_TO_REAL(PosAmp) * SIN( Ph )) + PosOffset;
		ServoCtrl.TargetTorque := 0;
		//ServoCtrl.PosTarget := OutRefP;
		(*Profile_CSP_DB(
	p_in:= gvl_io.Position_sp_test, 
	pold:= , 
	vold:= , 
	vcc:= 100, 
	acc:= 100, 
	Ts:= 0.001);*)
	
	
	(*
	Profile_CSP_DB(
	p_in:= DINT_TO_REAL(gvl_io.Position_sp_test), 
	pold:= gvl_io.pp, 
	vold:= gvl_io.pv, 
	vcc:= gvl_io.vcc_SP, 
	acc:= gvl_IO.acc_SP, 
	Ts:= 0.001, 
	pp=> gvl_io.pp, 
	pv=> gvl_io.pv);
		*)
		
		//ServoCtrl.PosTarget := gvl_io.Position_sp_test;
		ServoCtrl.PosTarget := REAL_TO_DINT(gvl_io.pp);
E_ModesOfOperation.ED_MO_Cyclic_sync_torque_mode:
		TorCmd_ds402  := TRUNC_INT( Amp * 1E6 / UDINT_TO_REAL(Motor_rated_torque0x6076));// TC*10e6/0x6076
		OutRef := TRUNC_INT( TorCmd_ds402 * SIN( Ph ));
		ServoCtrl.TargetTorque := OutRef;
E_ModesOfOperation.ED_MO_Cyclic_sync_velocity_mode:
		OutRefP := TRUNC( UDINT_TO_REAL(PosAmp) * SIN( Ph )) ;
		ServoCtrl.TargetTorque := 0;
		ServoCtrl.Target_velocity0x60FF := OutRefP;

END_CASE
ServoCtrl.ModeOfOperation := TO_SINT(Mode_of_operation);
END_METHOD

METHOD Restart : BOOL
VAR_INPUT
END_VAR
	nCycles   := 0;
	ind  :=0;
END_METHOD

END_FUNCTION_BLOCK

// ---- POUs/InitSDO_w.TcPOU
FUNCTION_BLOCK InitSDO_w
VAR_INPUT
//	bInit_Sdo_States : BOOL;
	sNetId     : T_AmsNetId;
	nSlaveAddr : UINT;
	ProfParams : Ds402_Params;

END_VAR
VAR_OUTPUT
	Sdo_States : ARRAY [0..10] OF CSdo_State ;
	bInitDone  : BOOL := FALSE;
	bError : bool := false;
END_VAR
VAR
	fbSdoWrite  : FB_EcCoESdoWrite;
	indSdo :   USINT :=0;
END_VAR

METHOD Init : BOOL
VAR_INPUT
END_VAR
//IF bInit_Sdo_States THEN
	Sdo_States[0].pBuf   	:= ADR(ProfParams.Abort_connection_option_code_0x6007);
    Sdo_States[0].nBufLen 	:=SIZEOF(ProfParams.Abort_connection_option_code_0x6007);
	Sdo_States[0].nIndex 	:=16#6007;
	Sdo_States[0].nSubIndex :=0;
	Sdo_States[0].bExecute := TRUE;
	
	Sdo_States[1].pBuf   	:= ADR(ProfParams.Postion_window0x6067);
    Sdo_States[1].nBufLen 	:=SIZEOF(ProfParams.Postion_window0x6067);
	Sdo_States[1].nIndex 	:=16#6067;
	Sdo_States[1].nSubIndex :=0;
	Sdo_States[1].bExecute := TRUE;
	
	
	Sdo_States[2].pBuf   	:= ADR(ProfParams.Position_window_time0x6068);
    Sdo_States[2].nBufLen 	:=SIZEOF(ProfParams.Position_window_time0x6068);
	Sdo_States[2].nIndex 	:=16#6068;
	Sdo_States[2].nSubIndex :=0;
	Sdo_States[2].bExecute := TRUE;

	Sdo_States[3].pBuf   	:= ADR(ProfParams.Interpolation_time_period0x60C2_1_period);
    Sdo_States[3].nBufLen 	:=SIZEOF(ProfParams.Interpolation_time_period0x60C2_1_period);
	Sdo_States[3].nIndex 	:=16#60C2;
	Sdo_States[3].nSubIndex :=1;
	Sdo_States[3].bExecute := TRUE;
//
	Sdo_States[4].pBuf   	:= ADR(ProfParams.Interpolation_time_period0x60C2_2_period);
    Sdo_States[4].nBufLen 	:=SIZEOF(ProfParams.Interpolation_time_period0x60C2_2_period);
	Sdo_States[4].nIndex 	:=16#60C2;
	Sdo_States[4].nSubIndex :=2;
	Sdo_States[4].bExecute := TRUE;
	
	
	
	(*
    Sdo_States[0].pBuf   	:= ADR(ProfParams_w.Interpolation_time_period0x60C2_2_period);
    Sdo_States[0].nBufLen 	:=SIZEOF(ProfParams_w.Interpolation_time_period0x60C2_2_period);
	Sdo_States[0].nIndex 	:=16#60C2;
	Sdo_States[0].nSubIndex :=2;
	Sdo_States[0].bExecute := TRUE;
*)
(*
	Sdo_States[0].pBuf   	:= ADR(ProfParams_w.Postion_window0x6067);
    Sdo_States[0].nBufLen 	:=SIZEOF(ProfParams_w.Postion_window0x6067);
	Sdo_States[0].nIndex 	:=16#6067;
	Sdo_States[0].nSubIndex :=0;
	Sdo_States[0].bExecute := TRUE;
*)
	
	//	bInit_Sdo_States:= FALSE;
	bInitDone:=FALSE;

//END_IF
END_METHOD

METHOD writeSDO : BOOL
VAR_INPUT
END_VAR
IF Sdo_States[indSdo].nBufLen > 0 THEN
	fbSdoWrite(tTimeout:= T#1.0S , sNetId:= sNetId,nSlaveAddr :=nSlaveAddr,
			nIndex:=Sdo_States[indSdo].nIndex,
 			nSubIndex :=Sdo_States[indSdo].nSubIndex,
	 		pSrcBuf:= Sdo_States[indSdo].pBuf, cbBufLen:=Sdo_States[indSdo].nBufLen,
			bExecute:=Sdo_States[indSdo].bExecute);
	IF NOT fbSdoWrite.bBusy THEN
		Sdo_States[indSdo].bExecute := FALSE;
		IF NOT fbSdoWrite.bError THEN 
			(* read successful *)
			Sdo_States[indSdo].bError := FALSE;
			Sdo_States[indSdo].nErrId := 0;
		ELSE 
			(* read failed *)
			Sdo_States[indSdo].bError := fbSdoWrite.bError;
			Sdo_States[indSdo].nErrId := fbSdoWrite.nErrId;
		END_IF
		fbSdoWrite(bExecute:=Sdo_States[indSdo].bExecute);
		bError := bError OR Sdo_States[indSdo].bError;
		indSdo := indSdo+1;
	END_IF
ELSE
	bInitDone:= TRUE;
END_IF
END_METHOD

END_FUNCTION_BLOCK

// ---- POUs/InitSDO.TcPOU
FUNCTION_BLOCK InitSDO
VAR_INPUT
//	bInit_Sdo_States : BOOL;
	sNetId     : T_AmsNetId;
	nSlaveAddr : UINT;

END_VAR
VAR_OUTPUT
	Sdo_States : ARRAY [0..10] OF CSdo_State ;
	bInitDone  : BOOL := FALSE;
	ProfParams : Ds402_Params;
	bError : BOOL:=FALSE;
END_VAR
VAR
	fbSdoRead  : FB_EcCoESdoRead;
	indSdo :   USINT :=0;
END_VAR

METHOD Init : BOOL
VAR_INPUT
END_VAR
//IF bInit_Sdo_States THEN
	Sdo_States[0].pBuf   	:= ADR(ProfParams.vendorId_0x1081_1);
    Sdo_States[0].nBufLen 	:=SIZEOF(ProfParams.vendorId_0x1081_1);
	Sdo_States[0].nIndex 	:=16#1018;
	Sdo_States[0].nSubIndex :=1;

	Sdo_States[1].pBuf   	:= ADR(ProfParams.Abort_connection_option_code_0x6007);
    Sdo_States[1].nBufLen 	:=SIZEOF(ProfParams.Abort_connection_option_code_0x6007);
	Sdo_States[1].nIndex 	:=16#6007;
	Sdo_States[1].nSubIndex :=0;

	Sdo_States[2].pBuf   	:= ADR(ProfParams.Motor_rated_torque0x6076);
    Sdo_States[2].nBufLen 	:=SIZEOF(ProfParams.Motor_rated_torque0x6076);
	Sdo_States[2].nIndex 	:=16#6076;
	Sdo_States[2].nSubIndex :=0;
	

	Sdo_States[3].pBuf   	:= ADR(ProfParams.Position_window_time0x6068);
    Sdo_States[3].nBufLen 	:=SIZEOF(ProfParams.Position_window_time0x6068);
	Sdo_States[3].nIndex 	:=16#6068;
	Sdo_States[3].nSubIndex :=0;
	
	//
	Sdo_States[4].pBuf   	:= ADR(ProfParams.Torque_slope0x6087);
    Sdo_States[4].nBufLen 	:=SIZEOF(ProfParams.Torque_slope0x6087);
	Sdo_States[4].nIndex 	:=16#6087;
	Sdo_States[4].nSubIndex :=0;
//

//
	Sdo_States[5].pBuf   	:= ADR(ProfParams.Interpolation_time_period0x60C2_1_period);
    Sdo_States[5].nBufLen 	:=SIZEOF(ProfParams.Interpolation_time_period0x60C2_1_period);
	Sdo_States[5].nIndex 	:=16#60C2;
	Sdo_States[5].nSubIndex :=1;
//
	Sdo_States[6].pBuf   	:= ADR(ProfParams.Interpolation_time_period0x60C2_2_period);
    Sdo_States[6].nBufLen 	:=SIZEOF(ProfParams.Interpolation_time_period0x60C2_2_period);
	Sdo_States[6].nIndex 	:=16#60C2;
	Sdo_States[6].nSubIndex :=2;



	
//	bInit_Sdo_States:= FALSE;
	bInitDone:=FALSE;

//END_IF
END_METHOD

METHOD readSDO : BOOL
VAR_INPUT
END_VAR
IF Sdo_States[indSdo].nBufLen > 0 THEN
	fbSdoRead(sNetId:= sNetId,nSlaveAddr :=nSlaveAddr, nIndex:=Sdo_States[indSdo].nIndex,
 			nSubIndex :=Sdo_States[indSdo].nSubIndex,
	 		pDstBuf:= Sdo_States[indSdo].pBuf, cbBufLen:=Sdo_States[indSdo].nBufLen,bExecute:=Sdo_States[indSdo].bExecute);
	IF NOT fbSdoRead.bBusy THEN
		Sdo_States[indSdo].bExecute := FALSE;
		IF NOT fbSdoRead.bError THEN 
			(* read successful *)
			Sdo_States[indSdo].bError := FALSE;
			Sdo_States[indSdo].nErrId := 0;
		ELSE 
			(* read failed *)
			Sdo_States[indSdo].bError := fbSdoRead.bError;
			Sdo_States[indSdo].nErrId := fbSdoRead.nErrId;
		END_IF
		fbSdoRead(bExecute:=Sdo_States[indSdo].bExecute);
		bError := bError OR Sdo_States[indSdo].bError;
		indSdo := indSdo+1;
	END_IF
ELSE
	bInitDone:= TRUE;
END_IF
END_METHOD

END_FUNCTION_BLOCK

// ---- POUs/FB_PosTest.TcPOU
FUNCTION_BLOCK FB_PosTest
VAR_INPUT
	PosTargetR : DINT;
	PosTargetL : DINT;
END_VAR
VAR_OUTPUT
	ApplyPosTargetNow : BOOL :=FALSE;
	PosCmd : DINT;
	nCycles : DINT := 0;
END_VAR
VAR
	eStateMachine		: E_PosTest := E_PosTest.Idle_init;
	inWindow : BOOL := TRUE;
	waitApplyPosTargetNow : UDINT;
END_VAR

METHOD Execute : BOOL
VAR_INPUT
END_VAR
VAR
END_VAR
CASE eStateMachine OF
	E_PosTest.Idle_init:
		ApplyPosTargetNow := FALSE;
		waitApplyPosTargetNow:=1000;
		IF Ds402.StatusWord_Bits.SwitchOn THEN
			eStateMachine := E_PosTest.Idle_start;
		END_IF
	E_PosTest.Idle_start:
	waitApplyPosTargetNow:=waitApplyPosTargetNow-1;
	IF waitApplyPosTargetNow =0 THEN
		eStateMachine := E_PosTest.GoToNextState_levelHi;
	END_IF
	
	E_PosTest.GoToNextState_levelHi:
	nCycles:=nCycles+1;
		PosCmd := PosTargetR;
		ApplyPosTargetNow := TRUE;//waitApplyPosTargetNow:=1000;
		eStateMachine := E_PosTest.MovingTo_levelHi;
		inWindow := TRUE;
	E_PosTest.MovingTo_levelHi:
		//waitApplyPosTargetNow:=waitApplyPosTargetNow-1;
		//IF  waitApplyPosTargetNow=0  THEN
		//ApplyPosTargetNow := FALSE;
		//END_IF
			IF Ds402.StatusWord_Bits.SetPointAck THEN
				ApplyPosTargetNow := FALSE;
			END_IF

		IF NOT Ds402.StatusWord_Bits.TargetReached THEN
			inWindow := FALSE;
		END_IF
		IF  Ds402.StatusWord_Bits.TargetReached AND NOT inWindow THEN
			eStateMachine := E_PosTest.GoToNextState_levelLo;
		END_IF

	E_PosTest.GoToNextState_levelLo:
		PosCmd := PosTargetL;
		ApplyPosTargetNow := TRUE;//waitApplyPosTargetNow:=1000;
		eStateMachine := E_PosTest.MovingTo_levelLo;
		inWindow := TRUE;
	E_PosTest.MovingTo_levelLo:
		//waitApplyPosTargetNow:=waitApplyPosTargetNow-1;
		//IF  waitApplyPosTargetNow=0  THEN
		//	ApplyPosTargetNow := FALSE;
		//END_IF
		IF Ds402.StatusWord_Bits.SetPointAck THEN
			ApplyPosTargetNow := FALSE;
		END_IF

		IF NOT Ds402.StatusWord_Bits.TargetReached THEN
			inWindow := FALSE;
		END_IF
		IF  Ds402.StatusWord_Bits.TargetReached AND NOT inWindow THEN
			eStateMachine := E_PosTest.GoToNextState_levelHi;
		END_IF
		
END_CASE


ServoCtrl.PosTarget := PosCmd;
ServoCtrl.TargetTorque := 0;
ServoCtrl.ModeOfOperation := TO_SINT(E_ModesOfOperation.ED_MO_Profile_position_mode);
END_METHOD

METHOD Restart : BOOL
VAR_INPUT
END_VAR
	eStateMachine		  := E_PosTest.Idle_init;
	inWindow   := TRUE;
	nCycles    :=  0;
END_METHOD

END_FUNCTION_BLOCK

// ---- POUs/FB_GetMasterTs.TcPOU
FUNCTION_BLOCK FB_GetMasterTs
VAR_INPUT
END_VAR
VAR_OUTPUT
	MasterTsUsec: INT :=0;
END_VAR
VAR
	prevTaskTime : ULINT;//100 ns
	nowTaskTime  : ULINT;//100 ns
	nCycles : ULINT :=0;
END_VAR

prevTaskTime := nowTaskTime;
nowTaskTime  := F_GetTaskTime();
IF nCycles>0 THEN
MasterTsUsec := ULINT_TO_INT( (nowTaskTime-prevTaskTime))/10;
END_IF
nCycles := nCycles+1;

END_FUNCTION_BLOCK

// ---- Function Blocks/FB_Sequence.TcPOU
FUNCTION_BLOCK FB_Sequence
VAR_INPUT
END_VAR
VAR_OUTPUT
END_VAR
VAR
	UP_Pause_ton: TON;
	tonReset_Long: TON;
	tonGripper_Open_error: TON;
	tonGropper_Close_Error: TON;
	tonEnable_Motor : TON;
	tonDesable_Motor : TON; 
	tonOneSensorError : TON;
	tonHomingError : TON;
	tonHomingStepDelay : TON;
	tonUserDelay : TON;
	tonMotionError : TON;
	tonLogTimer : TON;
		
	Always_ON :BOOL;
	Delay : BOOL;
	i , a , count: INT;
	Motor_curr_sum : REAL;
	

	
END_VAR

Always_ON := TRUE;
Delay := FALSE;


IF NOT gvl_IO.FirstScan 
	THEN
	gvl_io.qxActuator_1 := FALSE;
	gvl_IO.qxActuator_2 := FALSE;	
	gvl_io.Position_PV_Diff := 0 ;
	gvl_io.Position_sp_test := servoctrl.Position;	
	gvl_IO.FirstScan := TRUE;
END_IF


// Emergancy Stop 
IF NOT gvl_io.ixEmergancy_Stop
	THEN
	gvl_io.qxActuator_1 := FALSE;
	gvl_IO.qxActuator_2 := FALSE;
	gvl_io.Gripper_Close_cmd := FALSE;
	gvl_IO.Gripper_Open_cmd := FALSE;
	gvl_io.Gripper_step := 0;
	gvl_io.tonHomingStepDelay_IN := FALSE;
	gvl_io.tonHomingError_IN := FALSE;
	gvl_io.Step := 0;
	gvl_io.Homing_cmd := FALSE;
	gvl_io.Position_sp_test := servoctrl.Position;	
	gvl_io.tonHomingError_IN := FALSE;
	
END_IF


// Password

tonUserDelay(IN:= gvl_io.Password_IN = gvl_io.Password, PT:= T#5M , Q=> , ET=> );

IF tonUserDelay.Q 
	THEN
	gvl_io.Password_IN := 0;
END_IF


//********* Calculation MOTOR PARAMETRS***** 
(*
gvl_io.Position_PV := servoctrl.Position / (46603  *124  );
gvl_io.vcc_SP := gvl_io.Speed_SP * (46603  * 124 );

*)

gvl_io.Position_PV := servoctrl.Position / (46603  *124  );


IF GVL_IO.Step >= 0 
	AND GVL_IO.Step  < 700
	THEN
	gvl_io.vcc_SP := gvl_io.Speed_SP * (46603  * 124 );
	
	ELSIF
		 GVL_IO.Step  > 1000		 
		 THEN
		 gvl_io.vcc_SP := gvl_io.Speed_SP_slow * (46603  * 124 );
END_IF

gvl_io.Motor_I_PV := (DINT_TO_REAL(servoctrl.ActualCurrent) / 100 ) *2;
IF gvl_io.Motor_I_PV < 0 
	THEN gvl_io.Motor_I_PV := gvl_io.Motor_I_PV * (-1);
END_IF


// Change Accseleration bitwin Posoions
IF gvl_io.Homing_OK AND GVL_IO.Step> 1000 
	THEN
	gvl_io.acc_SP := gvl_io.Accseleration_SP_slow * (46603  * 124 );
	ELSIF gvl_io.Homing_OK AND GVL_IO.Step < 1000
		THEN			
			IF gvl_io.Position_PV_HMI > gvl_io.Position_UP_A_SP
				THEN
				gvl_io.acc_SP := gvl_io.Accseleration_A_SP * (46603 *124);
			ELSIF 
				gvl_io.Position_PV_HMI < gvl_io.Position_DN_A_SP
				THEN
				gvl_io.acc_SP := gvl_io.Accseleration_A_SP * (46603 *124);
			ELSE
				gvl_io.acc_SP := gvl_io.Accseleration_SP * (46603 *124);	
			END_IF
		
END_IF



IF servoctrl.ActualCurrent < 0 THEN 
	servoctrl.ActualCurrent := servoctrl.ActualCurrent * (-1) ;
END_IF

// MAnual command Go from HMI -  calculation Parametrs 
IF gvl_io.Homing_OK AND gvl_io.GO_TO_cmd THEN
	gvl_io.Position_sp_test := (gvl_io.Position_SP * 46603  *124) +  (gvl_io.Position_PV_Diff);
END_IF

// Positon_PV_HMI
gvl_io.Position_PV_HMI := (servoctrl.Position - gvl_io.Position_PV_Diff )/ (46603  *124  ) ;



IF GVL_IO.ixEmergancy_Stop AND GVL_IO.Enable
	AND NOT GVL_IO.Emergancy_Error
	THEN
	GVL_IO.Emergancy_OK := TRUE;
	ELSIF NOT GVL_IO.ixEmergancy_Stop
		THEN
		GVL_IO.Emergancy_OK := FALSE;	
		gvl_io.Enable_motor_cmd := FALSE;		
END_IF
//Emergancy Error
IF NOT GVL_IO.ixEmergancy_Stop 
	THEN 
	GVL_IO.Emergancy_Error := TRUE;	
END_IF

//Enable STO to Drive motor
GVL_IO.qxSTO_toDrive := Gvl_io.Enable;


// Ton TIMERS 
tonEnable_Motor(IN:= gvl_io.Enable_motor_cmd, PT:=T#500MS , Q=> , ET=> );
tonDesable_Motor(IN:= NOT gvl_io.Enable_motor_cmd, PT:=T#500MS , Q=> , ET=> );

// ******  Desable MOTOR *****
// close Breaks
IF NOT gvl_io.Enable_motor_cmd
	THEN gvl_io.qxBrakeOpen := FALSE;
END_IF
// desable  motor
IF NOT gvl_io.Enable_motor_cmd 
	AND tonDesable_Motor.Q	
	THEN
	gvl_io.Enable := FALSE;
END_IF


// Motor not ENABLE 
IF NOT gvl_io.Enable
	THEN 
	gvl_io.Position_sp_test := servoctrl.Position;
END_IF


// ****** MOTOR Limits *****
IF gvl_io.Position_PV_HMI >= gvl_io.Motor_Limit_UP
	OR gvl_io.Position_PV_HMI <= gvl_io.Motor_Limit_DN
	THEN
	gvl_io.Enable := FALSE;
END_IF


	
// ****** UP position Limits ****
IF gvl_io.Position_UP_SP >= gvl_io.Motor_Limit_UP - 1 
	THEN
	gvl_io.Position_UP_SP := gvl_io.Motor_Limit_UP - 1;	

ELSIF gvl_io.Position_UP_SP <= gvl_io.Motor_Limit_DN + 1 
	THEN 
	gvl_io.Position_UP_SP := gvl_io.Motor_Limit_DN + 1;		
END_IF


// ****** DN position Limits ****
IF gvl_io.Position_DN_SP <= gvl_io.Motor_Limit_DN + 1 
	THEN
	gvl_io.Position_DN_SP := gvl_io.Motor_Limit_DN + 1;	
ELSIF 	gvl_io.Position_DN_SP >= gvl_io.Motor_Limit_UP - 1 
	THEN
	gvl_io.Position_DN_SP := gvl_io.Motor_Limit_UP - 1;
END_IF




// ****** Enable MOTOR ***** 
//enable motor
IF gvl_io.Enable_motor_cmd
	THEN
	gvl_io.Enable := TRUE;
END_IF

IF gvl_io.Enable_motor_cmd
	AND tonEnable_Motor.Q
	THEN
	gvl_io.qxBrakeOpen := TRUE;
END_IF


// Error global
GVL_IO.Error := GVL_IO.Gripper_Open_Error 
				OR GVL_IO.Gripper_Close_Error 
				OR gvl_io.SensorLock_Error 
				OR gvl_io.Homing_Error 
				OR gvl_io.Motor_Error;

(*// TON MOTION ERROR 
tonMotionError(IN:= gvl_io.Homing_OK AND gvl_io.Step <> 0 AND gvl_io.tonMotionError_IN , PT:= T#5S , Q=> , ET=> );

gvl_io.tonMotionError_IN := servoCtrl.Position > (servoCtrl.PosTarget + 100)
							OR servoCtrl.Position < (servoCtrl.PosTarget - 100);

IF 
(servoCtrl.Position - gvl_io.pp > 32000
OR servoCtrl.Position - gvl_io.pp < 32000)
THEN

*)


// ********* Motor Error ******  ERROR POSITION ****

IF gvl_io.Homing_OK 
AND ( servoCtrl.StatusWord.3 
	OR  ABS(servoCtrl.Position - REAL_TO_DINT(gvl_io.pp)) > 23100000)
		THEN
	gvl_io.Motor_Error := TRUE;
	gvl_io.Enable_motor_cmd := FALSE;
	
END_IF
	
 
//Reset Errors
IF GVL_IO.Reset 
	THEN
	GVL_IO.Gripper_Open_Error := FALSE;
	GVL_IO.Gripper_Close_Error := FALSE;
	GVL_IO.Emergancy_Error := FALSE;
	gvl_io.SensorLock_Error := FALSE;
	gvl_io.Homing_Error := FALSE;
	gvl_io.Motor_Error := FALSE;
	gvl_io.Log_CloseFile_cmd := FALSE;	
END_IF

//TON Reset Long 
tonReset_Long(IN:= GVL_IO.Reset, PT:= T#5S, Q=> , ET=> );
IF tonReset_Long.Q
	THEN
	GVL_IO.Step := 0; 
	GVL_IO.UP_pause_in := FALSE;
	GVL_IO.qxClose_Gripper := FALSE;
	GVL_IO.qxOpen_Gripper := FALSE;
	GVL_IO.GO_TO_cmd := FALSE;	
	gvl_io.tonHomingError_IN := FALSE;
	gvl_io.Log_CloseFile_cmd := FALSE;
	
END_IF


// TON UP Pause 
UP_Pause_ton(IN:= GVL_IO.UP_pause_in, PT:= T#1S, Q=> , ET=> );

gvl_io.TwoSensorLock := gvl_io.ixGripperLock_1 AND gvl_io.ixGripperLock_2;


// TON Homing Error
tonHomingError(IN:= gvl_io.tonHomingError_IN, PT:= T#60S , Q=> , ET=> );
IF tonHomingError.Q
	THEN
	gvl_io.Position_sp_test := servoctrl.Position;
	gvl_io.Step := 0 ;
	gvl_io.Homing_cmd := FALSE;
	gvl_io.Enable_motor_cmd := FALSE;
	gvl_io.Homing_Error := TRUE;
	gvl_io.tonHomingError_IN := FALSE;	 
END_IF

// TON HOMING STEP DELAY 
tonHomingStepDelay(IN:= gvl_io.tonHomingStepDelay_IN , PT:= gvl_io.tonHomingStepDelay_SP, Q=> , ET=> );



//	STOP PB from HMI
IF (gvl_io.Stop 
	OR GVL_IO.Error)
	AND GVL_IO.Step <> 0 
	THEN
	gvl_io.Position_sp_test := servoctrl.Position;
	GVL_IO.Step := 0;
	GVL_IO.Start := FALSE;
END_IF


// Ready for Start
GVL_IO.Ready_for_start := GVL_IO.Emergancy_OK 
						AND GVL_IO.Homing_OK 
						
						//AND GVL_IO.ixHome_Position 
						AND NOT GVL_IO.Error;


// Sequence
CASE GVL_IO.Step OF 
	
	0: //
	i := 0;
	gvl_io.New_CSV_cmd := FALSE;
	IF GVL_IO.Ready_for_start 
		AND GVL_IO.Position_PV_HMI <> GVL_IO.Position_UP_SP
		AND GVL_IO.Motor_UP 
		THEN		
		GVL_IO.Step := 10;
	ELSIF GVL_IO.Ready_for_start AND GVL_IO.ixHome_Position
		AND GVL_IO.test_Gripper_close_OK
		AND GVL_IO.test_Gripper_open_OK
		AND GVL_IO.test_motor_sldown_ok
		AND GVL_IO.test_motor_slUP_ok
		AND GVL_IO.test_Insert_OK
		AND GVL_IO.test_slowCycle_OK
		AND GVL_IO.ATP_start_cmd AND GVL_RunLog.SN_valid	// no valid SN, no ATP start
		THEN
		GVL_IO.Step := 210;
		GVL_IO.Cycle_PV := 0;
	ELSIF GVL_IO.Ready_for_start AND GVL_IO.ixHome_Position
		AND GVL_IO.test_Gripper_close_OK
		AND GVL_IO.test_Gripper_open_OK
		AND GVL_IO.test_motor_sldown_ok
		AND GVL_IO.test_motor_slUP_ok
		AND GVL_IO.test_Insert_OK
		AND GVL_IO.Slow_cycle_cmd
		THEN 
		GVL_IO.Step := 1210;
		GVL_IO.Cycle_PV := 0;						
	ELSIF GVL_IO.Ready_for_start 
		AND GVL_IO.Position_PV_HMI <> GVL_IO.Position_DN_SP
		AND GVL_IO.Motor_DN
		THEN
		GVL_IO.Step := 110;
	ELSIF GVL_IO.Ready_for_start AND GVL_IO.ixHome_Position
		AND GVL_IO.Cycle_SP > 0
		AND GVL_IO.Start
		THEN
		GVL_IO.Step := 210;
		GVL_IO.Cycle_PV := 0;
	ELSIF GVL_IO.Homing
		AND gvl_io.Emergancy_OK 
		THEN
		GVL_IO.Step := 700;
	ELSIF GVL_IO.Ready_for_start 
		AND GVL_IO.Position_PV_HMI <> GVL_IO.Position_UP_SP
		AND GVL_IO.Motor_UP_slow_cmd
		THEN		
		GVL_IO.Step := 1010;
	ELSIF GVL_IO.Ready_for_start 
		AND GVL_IO.Position_PV_HMI <> GVL_IO.Position_DN_SP
		AND GVL_IO.Motor_DN_slow_cmd
		THEN
		GVL_IO.Step := 1110;		
	END_IF

	
	10:		//Motor UP command - write parameters
	gvl_io.Position_sp_test := (GVL_IO.Position_UP_SP * 46603  * 124) + (gvl_io.Position_PV_Diff);
	GVL_IO.Position_UP_SP_HL := (GVL_IO.Position_UP_SP) + 1;
	GVL_IO.Position_UP_SP_LL := (GVL_IO.Position_UP_SP) - 1;
	GVL_IO.Step := 20;
	
	20:		//Motor UP command - Wait finish motion
	IF GVL_IO.Position_PV_HMI = GVL_IO.Position_UP_SP
		OR (GVL_IO.Position_PV_HMI >= gvl_io.Position_UP_SP_LL AND GVL_IO.Position_PV_HMI <= gvl_io.Position_UP_SP_HL )
		THEN
		GVL_IO.Step := 0;
	END_IF
	
	110:	//MOtor DN command - write parameters
	gvl_io.Position_sp_test := (GVL_IO.Position_DN_SP * 46603  *124) +  (gvl_io.Position_PV_Diff);
	GVL_IO.Position_DN_SP_HL := (GVL_IO.Position_DN_SP) + 1;
	GVL_IO.Position_DN_SP_LL := (GVL_IO.Position_DN_SP) - 1;
	GVL_IO.Step := 120;
	
	120:	//Motor UP command - Wait finish motion
	IF GVL_IO.Position_PV_HMI = GVL_IO.Position_DN_SP
		OR (GVL_IO.Position_PV_HMI >= gvl_io.Position_DN_SP_LL AND GVL_IO.Position_PV_HMI <= gvl_io.Position_DN_SP_HL )
		THEN
		GVL_IO.Step := 0;
	END_IF
	
	210:	//Cycle -  open gripper 
	FOR a := 1 TO 500 DO 
		gvl_io.Position_PV_mem[a] := 0;
		gvl_io.Motor_I_mem[a] := 0.0;
	END_FOR
	gvl_io.Motor_I_MAX := 0.0;
	gvl_io.Motor_I_AVR := 0.0;
	
	GVL_IO.Gripper_Open_cmd := TRUE;
	GVL_IO.Step := 220;
	//gvl_io.New_CSV_cmd := TRUE;
	gvl_io.Log_Data := TRUE;
	gvl_io.Log_nMode := 2;
	
	220:	//Cycle - wait feedback gripper opened
	IF GVL_IO.ixGripper_Unlock
		AND NOT GVL_IO.Gripper_Open_cmd
		THEN 		
		GVL_IO.Step := 230;
		gvl_io.Log_Data := FALSE;
	END_IF
	
	230:	//Cycle - write parameters
	gvl_io.Position_sp_test := (GVL_IO.Position_DN_SP * 46603  *124) +  (gvl_io.Position_PV_Diff);
	GVL_IO.Position_DN_SP_HL := (GVL_IO.Position_DN_SP) + 1;
	GVL_IO.Position_DN_SP_LL := (GVL_IO.Position_DN_SP) - 1;
	GVL_IO.Step := 240;
	
	240:	//Cycle - Wait finish motion
	IF GVL_IO.Position_PV_HMI = GVL_IO.Position_DN_SP
		OR (GVL_IO.Position_PV_HMI >= gvl_io.Position_DN_SP_LL AND GVL_IO.Position_PV_HMI <= gvl_io.Position_DN_SP_HL )
		THEN
		gvl_io.Log_Data := TRUE;
		gvl_io.Log_nMode := 4;
		GVL_IO.Step := 260;
	END_IF
	
	
	260:	//Cycle - close gripper
	GVL_IO.Gripper_Close_cmd := TRUE;
	GVL_IO.Step := 270;
	
	270:	//Cycle - wait gripper close
	IF GVL_IO.ixGripperLock_1
		AND GVL_IO.ixGripperLock_2
		AND NOT GVL_IO.Gripper_Close_cmd
		THEN		
		GVL_IO.Step := 280;
	END_IF
	
	
	280:	//Cycle - write parameters 	
	gvl_io.Position_sp_test := (GVL_IO.Position_UP_SP * 46603  *124) + (gvl_io.Position_PV_Diff);
	GVL_IO.Position_UP_SP_HL := (GVL_IO.Position_UP_SP) + 1;
	GVL_IO.Position_UP_SP_LL := (GVL_IO.Position_UP_SP) - 1;
	GVL_IO.Step := 290;
	
	290:	//Cycle - Wait finish UP motion
	IF GVL_IO.Position_PV_HMI = GVL_IO.Position_UP_SP
		OR (GVL_IO.Position_PV_HMI >= gvl_io.Position_UP_SP_LL AND GVL_IO.Position_PV_HMI <= gvl_io.Position_UP_SP_HL )
		THEN
		GVL_IO.Step := 310;
	END_IF
	
	310:	//Cycle - Pause 0.5 sec 
	GVL_IO.UP_pause_in := TRUE;
	IF up_pause_ton.Q 
		THEN
		GVL_IO.UP_pause_in := FALSE;
		GVL_IO.Step := 320;
	END_IF
	
	320:	//Cycle - MOtion DN Write parametrs	
	gvl_io.Position_sp_test := (GVL_IO.Position_DN_SP * 46603  *124) + (gvl_io.Position_PV_Diff);
	GVL_IO.Position_DN_SP_HL := (GVL_IO.Position_DN_SP) + 1;
	GVL_IO.Position_DN_SP_LL := (GVL_IO.Position_DN_SP) - 1;
	GVL_IO.Step := 330;
	
	330:	//Motor UP command - Wait finish motion
	IF GVL_IO.Position_PV_HMI = GVL_IO.Position_DN_SP
		OR (GVL_IO.Position_PV_HMI >= gvl_io.Position_DN_SP_LL AND GVL_IO.Position_PV_HMI <= gvl_io.Position_DN_SP_HL )
		THEN
		GVL_IO.Step := 350;
	END_IF
	
	350:	//Cycle -  open gripper 
	GVL_IO.Gripper_Open_cmd := TRUE;
	GVL_IO.Step := 360;
	
	360:	//Cycle - wait feedback gripper opened
	IF GVL_IO.ixGripper_Unlock
		AND NOT GVL_IO.Gripper_Open_cmd
		THEN 
		GVL_IO.Cycle_PV := GVL_IO.Cycle_PV + 1;
		GVL_IO.Step := 370;
	END_IF
	
	370:	//Cycle - Check cycle counters 
	IF GVL_IO.Cycle_PV < GVL_IO.Cycle_SP
		THEN
		GVL_IO.Step := 260;
	ELSIF
		GVL_IO.Cycle_PV >= GVL_IO.Cycle_SP
		THEN
		GVL_IO.Step := 400;			
	END_IF
	
	400:	//Cycle - TO Home position 	
	gvl_io.Position_sp_test := (GVL_IO.Position_UP_SP * 46603  *124) + (gvl_io.Position_PV_Diff);
	GVL_IO.Position_UP_SP_HL := (GVL_IO.Position_UP_SP) + 1;
	GVL_IO.Position_UP_SP_LL := (GVL_IO.Position_UP_SP) - 1;
	GVL_IO.Step := 410;
	
	410:	//Cycle - TO Home position - Wait finish UP motion
	IF GVL_IO.Position_PV_HMI = GVL_IO.Position_UP_SP
		OR (GVL_IO.Position_PV_HMI >= gvl_io.Position_UP_SP_LL AND GVL_IO.Position_PV_HMI <= gvl_io.Position_UP_SP_HL )
		THEN
		GVL_IO.Step := 430;
	END_IF
	
	430:	//Cycle - TO Home position - close gripper
	GVL_IO.Gripper_Close_cmd := TRUE;
	GVL_IO.Step := 440;
	
	440:	//Cycle - TO Home position - wait gripper close
	IF NOT GVL_IO.Gripper_Close_cmd 
		AND GVL_IO.ixGripperLock_1
		AND GVL_IO.ixGripperLock_2
		THEN
		GVL_IO.Step := 0;
		GVL_IO.Start := FALSE;
		gvl_io.Calc_log_cmd := TRUE;
		gvl_io.Log_CloseFile_cmd := TRUE;
		gvl_io.Lod_appendLine_cmd := FALSE;
		gvl_io.Log_Data:=FALSE;
	END_IF
	
	
	
	
	//***** HOUMING ******
	
	
	700:	//Write online parameters
	gvl_io.tonHomingError_IN := TRUE;
	gvl_io.Step := 710;
	
	710: 	//Check  Homing Sensor
	IF NOT gvl_io.ixHome_Position 
		THEN
		gvl_io.Homing_OK := FALSE;
		gvl_io.Step := 720;
		ELSE
			gvl_io.Step := 740;
			gvl_io.Homing_OK := FALSE;
	END_IF
	
	
	720: 	// Write Homing parametrs
	gvl_io.vcc_SP := 5 * (46603  * 124 );
	gvl_io.acc_SP := 5 * (46603 *124);
	gvl_io.Position_sp_test := (180 * 46603  *124) ;// - gvl_io.Position_PV_Diff - 100;
	gvl_io.Step := 730;
	
	
	730:	// Wait Homing Sensor 
	IF gvl_io.ixHome_Position 
		THEN
		gvl_io.Step := 740;	
	END_IF
	
	740: // Write homing parametrs
	
		gvl_io.Position_PV_Diff := 0 + servoctrl.Position;
		gvl_io.Position_PV_HMI := servoctrl.Position - gvl_io.Position_PV_Diff;
		gvl_io.Position_sp_test := servoctrl.Position;
		gvl_io.Step := 750;
		gvl_io.tonHomingStepDelay_IN := TRUE;
		gvl_io.tonHomingStepDelay_SP := T#3S;
				
	
		
	
	750: 	// Wait Delay , change Homing parametrs
	IF tonHomingStepDelay.Q
		THEN
		gvl_io.tonHomingStepDelay_IN := FALSE;
		gvl_io.vcc_SP := 4 * (46603  * 124 );
		gvl_io.acc_SP := 4 * (46603 *124);

		gvl_io.Position_sp_test := servoctrl.Position - (4 * 46603  *124) ;
		gvl_io.Step := 760;		
	END_IF
	
	
	760:	// wait moving to SP position
	IF servoctrl.Position < gvl_io.Position_sp_test +10
		AND servoctrl.Position > gvl_io.Position_sp_test -10
		THEN
		gvl_io.vcc_SP := 1 * (46603  * 124 );
		gvl_io.acc_SP := 2 * (46603 *124);
		gvl_io.Position_sp_test := gvl_io.Position_PV_Diff + 1000000;
		gvl_io.Step := 770;
	END_IF
	
	770:	// Wait Homing sensor
	IF gvl_io.ixHome_Position 
		THEN
		// Write homing parametrs	
		gvl_io.Position_PV_Diff := 0 + servoctrl.Position;
		gvl_io.Position_sp_test := servoctrl.Position;
		gvl_io.tonHomingStepDelay_IN := TRUE;
		gvl_io.tonHomingStepDelay_SP := T#500MS;
		gvl_io.Step := 780;		
	END_IF
	
	780:	// Wait Dalay 500 ms 
	IF tonHomingStepDelay.Q
		THEN
		gvl_io.tonHomingStepDelay_IN := FALSE; 
		gvl_io.Homing_OK := TRUE;
		gvl_io.Step := 0;	
		gvl_io.tonHomingError_IN := FALSE;
	END_IF
	
	
	
	// TEST SLOW SPEED 
	
	1010:		//Motor UP slow  command - write parameters
	
	
	gvl_io.vcc_SP := gvl_io.Speed_SP_slow * (46603  * 124 );
	gvl_io.acc_SP := gvl_io.Accseleration_SP_slow * (46603 *124);
	GVL_IO.Step := 1015;
	Delay := TRUE;
	
	
	1015: 	//write parameters
	IF NOT Delay
		THEN
			gvl_io.Position_sp_test := (GVL_IO.Position_UP_SP * 46603  * 124) + (gvl_io.Position_PV_Diff);
			GVL_IO.Position_UP_SP_HL := (GVL_IO.Position_UP_SP) + 1;
			GVL_IO.Position_UP_SP_LL := (GVL_IO.Position_UP_SP) - 1;
			GVL_IO.Step := 1020;
	END_IF;
	
	1020:		//Motor UP command - Wait finish motion
	IF GVL_IO.Position_PV_HMI = GVL_IO.Position_UP_SP
		OR (GVL_IO.Position_PV_HMI >= gvl_io.Position_UP_SP_LL AND GVL_IO.Position_PV_HMI <= gvl_io.Position_UP_SP_HL )
		THEN		
		gvl_io.test_motor_slUP_ok := TRUE;
		GVL_IO.Step := 0;
	END_IF
	
	1110:	//MOtor DN command - write parameters
	gvl_io.vcc_SP := gvl_io.Speed_SP_slow * (46603  * 124 );
	gvl_io.acc_SP := gvl_io.Accseleration_SP_slow * (46603 *124);
	GVL_IO.Step := 1115;
	Delay := TRUE;
	
	1115: 	//write parameters
	IF NOT Delay
		THEN
	
	gvl_io.Position_sp_test := (GVL_IO.Position_DN_SP * 46603  *124) +  (gvl_io.Position_PV_Diff);
	GVL_IO.Position_DN_SP_HL := (GVL_IO.Position_DN_SP) + 1;
	GVL_IO.Position_DN_SP_LL := (GVL_IO.Position_DN_SP) - 1;
	GVL_IO.Step := 1120;
	END_IF
	
	1120:	//Motor UP command - Wait finish motion
	IF GVL_IO.Position_PV_HMI = GVL_IO.Position_DN_SP
		OR (GVL_IO.Position_PV_HMI >= gvl_io.Position_DN_SP_LL AND GVL_IO.Position_PV_HMI <= gvl_io.Position_DN_SP_HL )
		THEN
		//gvl_io.Speed_SP := gvl_io.Speed_SP_mem ;
		//gvl_io.Accseleration_SP := gvl_io.Accseleration_SP_mem ;
		gvl_io.test_motor_sldown_ok := TRUE;
		GVL_IO.Step := 0;
	END_IF
	
////  ***************** SLOW CYCLE *****************

	1210:	//Cycle -  open gripper 
		
	
	
	FOR a := 1 TO 500 DO 
		gvl_io.Position_PV_mem[a] := 0;
		gvl_io.Motor_I_mem[a] := 0.0;
	END_FOR
	gvl_io.Motor_I_MAX := 0.0;
	gvl_io.Motor_I_AVR := 0.0;
	
	GVL_IO.Gripper_Open_cmd := TRUE;
	GVL_IO.Step := 1220;
	
	1220:	//Cycle - wait feedback gripper opened
	IF GVL_IO.ixGripper_Unlock
		AND NOT GVL_IO.Gripper_Open_cmd
		THEN 		
		GVL_IO.Step := 1230;
	END_IF
	
	1230:	//Cycle - write parameters
	
	gvl_io.Position_sp_test := (GVL_IO.Position_DN_SP * 46603  *124) +  (gvl_io.Position_PV_Diff);
	GVL_IO.Position_DN_SP_HL := (GVL_IO.Position_DN_SP) + 1;
	GVL_IO.Position_DN_SP_LL := (GVL_IO.Position_DN_SP) - 1;
	GVL_IO.Step := 1240;
	
	1240:	//Cycle - Wait finish motion
	IF GVL_IO.Position_PV_HMI = GVL_IO.Position_DN_SP
		OR (GVL_IO.Position_PV_HMI >= gvl_io.Position_DN_SP_LL AND GVL_IO.Position_PV_HMI <= gvl_io.Position_DN_SP_HL )
		THEN
		GVL_IO.Step := 1260;
	END_IF
	
	
	1260:	//Cycle - close gripper
	GVL_IO.Gripper_Close_cmd := TRUE;
	GVL_IO.Step := 1270;
	
	1270:	//Cycle - wait gripper close
	IF GVL_IO.ixGripperLock_1
		AND GVL_IO.ixGripperLock_2
		AND NOT GVL_IO.Gripper_Close_cmd
		THEN		
		GVL_IO.Step := 1280;
	END_IF
	
	
	1280:	//Cycle - write parameters 	
	gvl_io.Position_sp_test := (GVL_IO.Position_UP_SP * 46603  *124) + (gvl_io.Position_PV_Diff);
	GVL_IO.Position_UP_SP_HL := (GVL_IO.Position_UP_SP) + 1;
	GVL_IO.Position_UP_SP_LL := (GVL_IO.Position_UP_SP) - 1;
	GVL_IO.Step := 1290;
	
	1290:	//Cycle - Wait finish UP motion
	IF GVL_IO.Position_PV_HMI = GVL_IO.Position_UP_SP
		OR (GVL_IO.Position_PV_HMI >= gvl_io.Position_UP_SP_LL AND GVL_IO.Position_PV_HMI <= gvl_io.Position_UP_SP_HL )
		THEN
		GVL_IO.Step := 1310;
	END_IF
	
	1310:	//Cycle - Pause 0.5 sec 
	GVL_IO.UP_pause_in := TRUE;
	IF up_pause_ton.Q 
		THEN
		GVL_IO.UP_pause_in := FALSE;
		GVL_IO.Step := 1320;
	END_IF
	
	1320:	//Cycle - MOtion DN Write parametrs	
	gvl_io.Position_sp_test := (GVL_IO.Position_DN_SP * 46603  *124) + (gvl_io.Position_PV_Diff);
	GVL_IO.Position_DN_SP_HL := (GVL_IO.Position_DN_SP) + 1;
	GVL_IO.Position_DN_SP_LL := (GVL_IO.Position_DN_SP) - 1;
	GVL_IO.Step := 1330;
	
	1330:	//Motor UP command - Wait finish motion
	IF GVL_IO.Position_PV_HMI = GVL_IO.Position_DN_SP
		OR (GVL_IO.Position_PV_HMI >= gvl_io.Position_DN_SP_LL AND GVL_IO.Position_PV_HMI <= gvl_io.Position_DN_SP_HL )
		THEN
		GVL_IO.Step := 1350;
	END_IF
	
	1350:	//Cycle -  open gripper 
	GVL_IO.Gripper_Open_cmd := TRUE;
	GVL_IO.Step := 1360;
	
	1360:	//Cycle - wait feedback gripper opened
	IF GVL_IO.ixGripper_Unlock
		AND NOT GVL_IO.Gripper_Open_cmd
		THEN 
		GVL_IO.Cycle_PV := GVL_IO.Cycle_PV + 1;
		GVL_IO.Step := 1370;
	END_IF
	
	1370:	//Cycle - Check cycle counters 
(*	
IF GVL_IO.Cycle_PV < GVL_IO.Cycle_SP
		THEN
		GVL_IO.Step := 260;
	ELSIF
		GVL_IO.Cycle_PV >= GVL_IO.Cycle_SP
		THEN
		GVL_IO.Step := 400;			
	END_IF
	*)
	
	GVL_IO.Step := 1400;	
	
	1400:	//Cycle - TO Home position 	
	gvl_io.Position_sp_test := (GVL_IO.Position_UP_SP * 46603  *124) + (gvl_io.Position_PV_Diff);
	GVL_IO.Position_UP_SP_HL := (GVL_IO.Position_UP_SP) + 1;
	GVL_IO.Position_UP_SP_LL := (GVL_IO.Position_UP_SP) - 1;
	GVL_IO.Step := 1410;
	
	1410:	//Cycle - TO Home position - Wait finish UP motion
	IF GVL_IO.Position_PV_HMI = GVL_IO.Position_UP_SP
		OR (GVL_IO.Position_PV_HMI >= gvl_io.Position_UP_SP_LL AND GVL_IO.Position_PV_HMI <= gvl_io.Position_UP_SP_HL )
		THEN
		GVL_IO.Step := 1430;
	END_IF
	
	1430:	//Cycle - TO Home position - close gripper
	GVL_IO.Gripper_Close_cmd := TRUE;
	GVL_IO.Step := 1440;
	
	1440:	//Cycle - TO Home position - wait gripper close
	IF NOT GVL_IO.Gripper_Close_cmd 
		AND GVL_IO.ixGripperLock_1
		AND GVL_IO.ixGripperLock_2
		THEN
		GVL_IO.Step := 0;
		GVL_IO.Start := FALSE;
		GVL_IO.test_slowCycle_OK := TRUE;
		
	END_IF
	
	
	
	
	
	

END_CASE

///// ******* Posotion SP Limit *******
IF gvl_io.Position_SP  >= gvl_io.Motor_Limit_UP - 1 
	THEN
	gvl_io.Position_SP := gvl_io.Motor_Limit_UP - 1; 
	ELSIF 
		gvl_io.Position_SP <= gvl_io.Motor_Limit_DN + 1 
	THEN 
	gvl_io.Position_SP := gvl_io.Motor_Limit_DN + 1;
END_IF



// 		******** GRIPPER *************

// One Sensor lock not work 
tonOneSensorError(IN:= gvl_io.Gripper_step >0 AND ((gvl_io.ixGripperLock_1 AND NOT gvl_io.ixGripperLock_2) OR (NOT  gvl_io.ixGripperLock_1 AND gvl_io.ixGripperLock_2)) , PT:= T#2S , Q=> , ET=> );
IF tonOneSensorError.Q
	THEN
	gvl_io.SensorLock_Error := TRUE;
END_IF

//TON Gripper Open Error
tonGripper_Open_error(IN:= GVL_IO.Gripper_Open_cmd OR (gvl_io.Gripper_step >0 AND gvl_io.Gripper_step <=130), PT:= T#2S, Q=> , ET=> );
IF tonGripper_Open_error.Q
	THEN
		GVL_IO.Gripper_Open_Error := TRUE;
		GVL_IO.qxActuator_1 := FALSE;
		GVL_IO.qxActuator_2 := FALSE;
		GVL_IO.Gripper_Open_cmd  := FALSE;
		gvl_io.test_Gripper_open_OK := FALSE;
		gvl_io.Gripper_step := 0;
		gvl_io.Step := 0;
END_IF


//TON Gripper Close Error
tonGropper_Close_Error(IN:= GVL_IO.Gripper_Close_cmd OR (gvl_io.Gripper_step >=200 AND gvl_io.Gripper_step <=230) , PT:= T#2S , Q=> , ET=> );
IF tonGropper_Close_Error.Q
	THEN
		GVL_IO.Gripper_Close_Error := TRUE;
		GVL_IO.qxActuator_1 := FALSE;
		GVL_IO.qxActuator_2 := FALSE;
		GVL_IO.Gripper_Close_cmd  := FALSE;
		gvl_io.test_Gripper_close_OK := TRUE;
		gvl_io.Gripper_step := 0;
		gvl_io.Step := 0;		
END_IF

CASE GVL_IO.Gripper_step OF 
	
	0: 	// Wait command 
	IF gvl_io.Gripper_Open_cmd 
		AND NOT GVL_IO.Error
		THEN
			GVL_IO.Gripper_step := 100; // Open Gripper
		ELSIF gvl_io.Gripper_Close_cmd 
			AND NOT GVL_IO.Error
			THEN
			gvl_io.Gripper_step := 200; // Close Gripper
	END_IF
	
	100: 	//check sensor 
	IF gvl_io.ixGripper_Unlock
		THEN
			gvl_io.Gripper_Open_cmd := FALSE;
			gvl_io.Gripper_step := 0;
		ELSE
			gvl_io.Gripper_step := 110;
	END_IF
	
	
	110: 	//Open Gripper sequence
	gvl_io.qxActuator_1 := TRUE;
	gvl_io.qxActuator_2 := TRUE;
	gvl_io.Gripper_step := 120;
	
	120: 	// wait sensor 
	IF gvl_io.ixGripper_Unlock
		THEN
		gvl_io.qxActuator_1 := FALSE;
		gvl_io.qxActuator_2 := FALSE;
		gvl_io.Gripper_Open_cmd := FALSE;
		gvl_io.test_Gripper_open_OK := TRUE;
		gvl_io.Gripper_step := 0;
	END_IF
	
	
	
	200: 	//check sensor 
	IF gvl_io.ixGripperLock_1 AND gvl_io.ixGripperLock_2
		THEN
			gvl_io.Gripper_Close_cmd := FALSE;
			gvl_io.Gripper_step := 0;
		ELSE
			gvl_io.Gripper_step := 210;
	END_IF
	
	
	210: 	//Close Gripper sequence
	gvl_io.qxActuator_1 := FALSE;
	gvl_io.qxActuator_2 := TRUE;	
	gvl_io.Gripper_step := 220;
	
	220: 	// wait sensor 
	IF gvl_io.ixGripperLock_1 AND gvl_io.ixGripperLock_2
		THEN
		gvl_io.qxActuator_1 := FALSE;
		gvl_io.qxActuator_2 := FALSE;
		gvl_io.Gripper_Close_cmd := FALSE;
		gvl_io.test_Gripper_close_OK := TRUE;
		gvl_io.Gripper_step := 0;
	END_IF
	
	
END_CASE


//**************** LOG **************
tonLogTimer(IN:= gvl_io.tonLogTimer_IN AND NOT gvl_io.tonLogTimer_Q, PT:=T#100MS , Q=> gvl_io.tonLogTimer_Q, ET=> );
IF gvl_io.tonLogTimer_Q
	THEN
	gvl_io.Lod_appendLine_cmd := TRUE;
	i := i + 1;	
	IF i < 0 
		OR i > 500
		THEN
		i := 0;
	END_IF
END_IF



IF gvl_io.Step > 200 
	AND gvl_io.Step < 700
	AND GVL_IO.Cycle_PV >= (GVL_IO.Cycle_SP - 1)
	THEN
	gvl_io.tonLogTimer_IN := TRUE;
	ELSE
	gvl_io.tonLogTimer_IN := FALSE;	
END_IF

// 		Find MAX Motor current in last cycle 
IF gvl_io.tonLogTimer_IN
	AND gvl_io.Motor_I_MAX < gvl_io.Motor_I_PV
	THEN
	gvl_io.Motor_I_MAX := gvl_io.Motor_I_PV ;	
END_IF

// 		Calculation Average Motor Current in last cycle 
IF gvl_io.Lod_appendLine_cmd
	THEN
	gvl_io.Motor_I_mem[i] := gvl_io.Motor_I_PV;
	gvl_io.Position_PV_mem[i] := gvl_io.Position_PV_HMI;	
END_IF

IF gvl_io.Calc_log_cmd
	THEN
	count := 0;
	Motor_curr_sum := 0.0;
	FOR a := 1 TO 500 DO 	
	
		IF gvl_io.Motor_I_mem[a] > 0
			THEN
			Motor_curr_sum := Motor_curr_sum + gvl_io.Motor_I_mem[a];
			count := count + 1;
			
		END_IF	
	END_FOR
	
	gvl_io.Motor_I_AVR := Motor_curr_sum / INT_TO_REAL(count);	
	gvl_io.Calc_log_cmd := FALSE;
END_IF

END_FUNCTION_BLOCK

// ---- Function Blocks/Profil_CSP.TcPOU
FUNCTION_BLOCK Profil_CSP
VAR_INPUT
	p_in,pold,vold,vcc,acc,Ts : REAL;
	
END_VAR
VAR_OUTPUT
	pp, pv :REAL;
END_VAR
VAR
	 p, v , pTol, vTol , pnext, vnext : REAL;
	ProblemInverted : BOOL;
		


END_VAR

//FUNCTION [pp,pv] = SpeedOnlyProfilerA(p_in,pold,vold,vcc,acc,Ts);
//
// Difference left to this instance, no extra speed taken
p :=  ( p_in - pold ) ;

IF ( p < 0.0 ) THEN
    v := -vold ;
    p := -p ;
    ProblemInverted := TRUE ;
else
    v := vold  ;
    ProblemInverted := FALSE ;
END_IF

pTol := 0.5*acc*Ts*Ts;
vTol := acc*Ts;
IF( p < pTol AND ABS(v) < vTol ) THEN 
    pp := p_in ;
    pv := 0 ;
    return;
END_IF

vnext := v + acc*Ts;
IF vnext > SQRT(2*acc*p) THEN 
    vnext := SQRT(2*acc*p) ;
END_IF


IF vnext > vcc THEN
	vnext := vcc;
END_IF

pnext := 0.5 * Ts * ( v + vnext );

// We have the next speed and acceleration. Revert to frame
IF ProblemInverted THEN
	vnext := -vnext ;
    pnext := -pnext ;
END_IF

// Integrate speed and position references using the given acceleration
pnext := pold + pnext ;
pp := pnext ;
pv := vnext ;

END_FUNCTION_BLOCK

// ---- POUs/processStatusWord.TcPOU
FUNCTION processStatusWord : Ds402_SW
VAR_INPUT
	StatusWord : INT; 
END_VAR
VAR
	StatusWord_Bits : Ds402_SW;
END_VAR

// Process Status word
//StatusWord := ServoCtrl.StatusWord;

StatusWord_Bits.ReadyToSwitchOn := StatusWord.0;// = bitand(sw,1);
StatusWord_Bits.SwitchOn  := StatusWord.1;//= bitand(bitshift(sw,-1),1);
StatusWord_Bits.OperationEnabled  := StatusWord.2;// = bitand(bitshift(sw,-2),1);
StatusWord_Bits.Fault  := StatusWord.3;// = bitand(bitshift(sw,-3),1);
StatusWord_Bits.VoltageEnabled  := StatusWord.4;// = bitand(bitshift(sw,-4),1);
StatusWord_Bits.NoQuickStop  := StatusWord.5;// = bitand(bitshift(sw,-5),1);
StatusWord_Bits.SwitchOnDisabled  := StatusWord.6;// = bitand(bitshift(sw,-6),1);
StatusWord_Bits.Warning  := StatusWord.7;// = bitand(bitshift(sw,-7),1);
StatusWord_Bits.ManufacturerSpecific8  := StatusWord.8;// = bitand(bitshift(sw,-8),1);
StatusWord_Bits.Remote  := StatusWord.9;// = bitand(bitshift(sw,-9),1);
StatusWord_Bits.TargetReached  := StatusWord.10;// = bitand(bitshift(sw,-10),1);
StatusWord_Bits.InternalLimitActive  := StatusWord.11;// = bitand(bitshift(sw,-11),1);
StatusWord_Bits.OperationModeSpecific12to13  :=BIT_TO_INT(StatusWord.12) + 2*BIT_TO_INT(StatusWord.13)  ;// = bitand(bitshift(sw,-12),3);
StatusWord_Bits.ManufacturerSpecific14to15  := BIT_TO_INT(StatusWord.14) + 2*BIT_TO_INT(StatusWord.15)   ;// = bitand(bitshift(sw,-14),3);

StatusWord_Bits.SetPointAck := StatusWord.12;
StatusWord_Bits.FollowingError := StatusWord.13;

// Process control word
(*
if status == ST_WORD_SWITCH_ON_DISABLED
    TransitionList = [CTL_WORD_TRANSITION_SHUTDOWN,CTL_WORD_TRANSITION_SW_ON_ENA_OPER] ;
elseif status == ST_WORD_READY_TO_SWITCH_ON
    TransitionList = [CTL_WORD_TRANSITION_SW_ON_ENA_OPER] ;
elseif status == ST_WORD_SWITCHED_ON
    TransitionList = [CTL_WORD_TRANSITION_ENABLE_OPER] ;
elseif status == ST_WORD_OPERATION_ENABLED
    % Already oeration enabled - nothing to do
    return ;
*)
processStatusWord:= StatusWord_Bits;

END_FUNCTION

// ---- POUs/MotorOn.TcPOU
FUNCTION MotorOn : UINT
VAR_INPUT
	StatusWord_Bits : Ds402_SW;
	ApplyPosTargetNow : BOOL;
END_VAR
VAR
	ControlWord : UINT;
END_VAR

ControlWord := 16#000F;// default
IF (StatusWord_Bits.SwitchOnDisabled = TRUE ) THEN
	ControlWord := 6;
ELSE   	
		    IF (StatusWord_Bits.ReadyToSwitchOn = TRUE) THEN
			        ControlWord := 7;
			END_IF 
			
			IF (StatusWord_Bits.SwitchOn = TRUE) THEN
					ControlWord := 16#000F +   16#0020;//   change set immediately
			END_IF
			
END_IF
IF ApplyPosTargetNow THEN
	ControlWord.4 := 1; // New set point 
ELSE
	ControlWord.4 := 0; // clear point		
END_IF
IF	StatusWord_Bits.Fault THEN
	ControlWord.7 := 1;// clear fault
ELSE
	ControlWord.7 := 0;
END_IF
//ServoCtrl.ControlWord := ControlWord;
MotorOn := ControlWord;

END_FUNCTION

// ---- POUs/Prg_WritePersistentVars.TcPOU
PROGRAM Prg_WritePersistentVars
VAR
	//fb_FB_S_UPS: FB_S_UPS_CX51x0;
	fb_FB_S_UPS: FB_S_UPS_CX9020_U900;
	fb_FB_WritePersistentData: FB_WritePersistentData;
	
	_WritePersis: BOOL;
END_VAR


{IF defined (PLC)}
	fb_FB_S_UPS(
		sNetID:='' , 
		iPLCPort:=851 , 
		//iplPort:= , 
		tTimeout:= , 
		eUpsMode:=eSUPS_WrPersistData_Shutdown , 
		ePersistentMode:=SPDM_2PASS , 
		tRecoverTime:= , 
		bPowerFailDetect=> , 
		eState=> );
{ELSIF defined (Develop)}

{END_IF}
	
		

fb_FB_WritePersistentData(
	NETID:= , 
	PORT:= 851, 
	START:=_WritePersis , 
	TMOUT:= , 
	MODE:= , 
	BUSY=> , 
	ERR=> , 
	ERRID=> );

END_PROGRAM

// ---- POUs/Main_10ms.TcPOU
PROGRAM Main_10ms
VAR
END_VAR


Prg_GetClock();
Prg_logEvents();
OpenExplorer();

END_PROGRAM

// ---- POUs/Prg_GetClock.TcPOU
PROGRAM Prg_GetClock
VAR

(* Real Time Clock *)
	tRealTime				: DATE_AND_TIME;
	stSystemTime			: TimeStruct;

	sTime					: STRING[20];
	sDate					: STRING[20];
	sTimeWithMicroSec		: STRING[40];

	syncTimer 	: TON;
	fbGetLocalTime 	: NT_GetTime;
	fbRTC_EX2 	: RTC_EX2;
	presetTime 	: TimeStruct;
	syncTrigger 	: F_TRIG;
	bBusy 		: BOOL;
	bError 		: BOOL;
	nErrID 		: UDINT;
	temp1: DATE;
	temp2: TOD;
	NetId :STRING :='';
	bValid_RTCEX2 	: BOOL;
	nMicroseconds 	: DWORD;
	WeekOfYear: INT;
END_VAR

(*--------->Set Plc Clock<----------------*)

tRealTime:=SYSTEMTIME_TO_DT(stSystemTime);
temp1:=DT_TO_DATE(tRealTime);
temp2:=DT_TO_TOD(tRealTime);
sDate:=DATE_TO_STRING(temp1);
sDate:=DELETE(sDate,2,1);


sTime:=TOD_TO_STRING(temp2);
sTime:=DELETE(sTime,4,1);
sTimeWithMicroSec:=CONCAT(sTime,'.');
sTimeWithMicroSec:=CONCAT(sTimeWithMicroSec,DWORD_TO_STRING(nMicroseconds));




	syncTimer(IN:=NOT SyncTimer.Q , PT:=T#1s , Q=> , ET=> );

	fbGetLocalTime(
		NETID:='' ,
		START:=syncTimer.Q,
		TMOUT:=T#5s ,
		BUSY=>bBusy ,
		ERR=>bError ,
		ERRID=>nErrId ,
		TIMESTR=>presetTime );

	syncTrigger(CLK:=NOT bBusy
					 AND NOT bError , Q=> );
	fbRTC_EX2(
		EN:=syncTrigger.Q ,
		PDT:=presetTime ,
		PMICRO:=0 ,
		Q=>bValid_RTCEX2 ,
		CDT=>stSystemTime ,
		CMICRO=>nMicroseconds );

WeekOfYear:=F_GetWeekOfTheYear(tRealTime);

END_PROGRAM

// ---- POUs/Prg_logEvents.TcPOU
// Adapter between the run sequence and the run log module (RunLog\FB_RunLogger).
// FB_Sequence keeps raising the same commands it always did - Log_Data, Lod_appendLine_cmd,
// Log_CloseFile_cmd; how and where a run is written is decided in FB_RunLogger only.
PROGRAM Prg_logEvents
VAR
	fbRunLogger : FB_RunLogger;
END_VAR

GVL_RunLog.SN_valid := F_RunLogSnValid(GVL_RunLog.SN);

fbRunLogger(
	bStart := gvl_io.Log_Data,
	bRunActive := gvl_io.Step <> 0,
	bReset := gvl_io.Reset,
	sSN := GVL_RunLog.SN,
	bSnValid := GVL_RunLog.SN_valid,
	nCyclesSet := gvl_io.Cycle_SP,
	rCurrent := gvl_io.Motor_I_PV,
	nPosition := gvl_io.Position_PV_HMI,
	stNow := Prg_GetClock.stSystemTime,
	bAppend := gvl_io.Lod_appendLine_cmd,
	bClose := gvl_io.Log_CloseFile_cmd);

GVL_RunLog.State := fbRunLogger.sState;
GVL_RunLog.LastFile := fbRunLogger.sLastFile;
GVL_RunLog.LastError := fbRunLogger.sLastError;
GVL_RunLog.ErrorCount := fbRunLogger.nErrors;

END_PROGRAM

// ---- RunLog/FB_RunLogger.TcPOU
// Writes one run log per run in the AUT003-ELM-LOG/1 format (report-tool/docs/log-format.md).
//
// The whole log format lives here; the run sequence only raises bStart, bAppend and bClose,
// as it did for the old logger. Replace or edit this block without touching FB_Sequence.
//
// File life: <dir>\<YYYYMMDD-HHMMSS>_<SN>.tmp while the run is written; renamed to .log when
// the run completes (bClose). A run that stops early (bRunActive falls, or bReset) keeps its
// .tmp - the reader never touches a .tmp, so an incomplete run cannot reach a report.
// A run started without a valid SN is not logged at all (sLastError says so).
FUNCTION_BLOCK FB_RunLogger
VAR_INPUT
	bStart		: BOOL;			// rising edge: open a file for a new run
	bRunActive	: BOOL;			// falls while a file is open = the run was stopped
	bReset		: BOOL;			// abandon the open file, keep it as .tmp
	sSN			: STRING(32);
	bSnValid	: BOOL;
	nCyclesSet	: UDINT;		// Cycle_SP; the logged cycle is the last one
	rCurrent	: REAL;			// Motor_I_PV
	nPosition	: DINT;			// Position_PV_HMI
	stNow		: TIMESTRUCT;	// PLC clock, for the file name and the start stamp
END_VAR
VAR_IN_OUT
	bAppend		: BOOL;			// one sample is due; cleared here when taken
	bClose		: BOOL;			// the run completed; cleared here when taken
END_VAR
VAR_OUTPUT
	bFileOpen	: BOOL;
	sState		: STRING(40);
	sLastFile	: STRING(255);
	sLastError	: STRING(255);
	nErrors		: UDINT;
END_VAR
VAR CONSTANT
	{IF defined (Develop)}
		LOG_DIR		: STRING := 'C:\Users\user\Source\Repos\AUT003_ELM\Export\Logs';
	{ELSE}
		// On Windows CE only \Hard Disk is on the card; \Temp may be in RAM.
		LOG_DIR		: STRING := '\Hard Disk\Logs';
	{END_IF}
	FORMAT_ID	: STRING := 'AUT003-ELM-LOG/1';
	SAMPLE_MS	: UDINT := 100;		// FB_Sequence raises bAppend every 100 ms
END_VAR
VAR
	rtStart		: R_TRIG;
	fbCreateDir	: FB_CreateDir;
	fbOpen		: FB_FileOpen;
	fbWrite		: FB_FileWrite;
	fbClose		: FB_FileClose;
	fbRename	: FB_FileRename;
	hFile		: UINT;
	nStep		: INT;
	bCompleted	: BOOL;			// TRUE: close then rename; FALSE: close and keep the .tmp
	nSamples	: UDINT;
	sStamp		: STRING(20);	// YYYYMMDD-HHMMSS
	sStartIso	: STRING(20);	// YYYY-MM-DDTHH:MM:SS
	sTmpPath	: STRING(255);
	sLogPath	: STRING(255);
	sBuffer		: STRING(255);	// must not change while fbWrite is busy
END_VAR

rtStart(CLK := bStart);

CASE nStep OF
	0:	// idle; a sample or close request with no file open is simply taken
		sState := 'idle';
		bFileOpen := FALSE;
		bAppend := FALSE;
		bClose := FALSE;
		IF rtStart.Q THEN
			IF NOT bSnValid THEN
				sLastError := CONCAT('run not logged - no valid SN: ', sSN);
			ELSE
				sStamp := CONCAT(WORD_TO_STRING(stNow.wYear), RIGHT(CONCAT('0', WORD_TO_STRING(stNow.wMonth)), 2));
				sStamp := CONCAT(sStamp, RIGHT(CONCAT('0', WORD_TO_STRING(stNow.wDay)), 2));
				sStamp := CONCAT(sStamp, '-');
				sStamp := CONCAT(sStamp, RIGHT(CONCAT('0', WORD_TO_STRING(stNow.wHour)), 2));
				sStamp := CONCAT(sStamp, RIGHT(CONCAT('0', WORD_TO_STRING(stNow.wMinute)), 2));
				sStamp := CONCAT(sStamp, RIGHT(CONCAT('0', WORD_TO_STRING(stNow.wSecond)), 2));
				// YYYYMMDD-HHMMSS -> YYYY-MM-DDTHH:MM:SS
				sStartIso := CONCAT(CONCAT(LEFT(sStamp, 4), '-'), MID(sStamp, 2, 5));
				sStartIso := CONCAT(CONCAT(sStartIso, '-'), MID(sStamp, 2, 7));
				sStartIso := CONCAT(CONCAT(sStartIso, 'T'), MID(sStamp, 2, 10));
				sStartIso := CONCAT(CONCAT(sStartIso, ':'), MID(sStamp, 2, 12));
				sStartIso := CONCAT(CONCAT(sStartIso, ':'), MID(sStamp, 2, 14));
				sTmpPath := CONCAT(CONCAT(CONCAT(LOG_DIR, '\'), sStamp), CONCAT('_', sSN));
				sLogPath := CONCAT(sTmpPath, '.log');
				sTmpPath := CONCAT(sTmpPath, '.tmp');
				nSamples := 0;
				bCompleted := FALSE;
				sState := 'opening';
				nStep := 10;
			END_IF
		END_IF

	10:	// the folder may already exist; an error here is not fatal, the open below decides
		fbCreateDir(sNetId := '', sPathName := LOG_DIR, bExecute := TRUE, tTimeout := T#5S);
		IF NOT fbCreateDir.bBusy THEN
			fbCreateDir(bExecute := FALSE);
			nStep := 20;
		END_IF

	20:	// binary: the $R$N line ends are written as they are
		fbOpen(sNetId := '', sPathName := sTmpPath, nMode := FOPEN_MODEWRITE OR FOPEN_MODEBINARY,
			ePath := PATH_GENERIC, bExecute := TRUE, tTimeout := T#5S);
		IF NOT fbOpen.bBusy THEN
			IF fbOpen.bError THEN
				sLastError := CONCAT('cannot create ', sTmpPath);
				nErrors := nErrors + 1;
				nStep := 0;
			ELSE
				hFile := fbOpen.hFile;
				bFileOpen := TRUE;
				sBuffer := CONCAT(CONCAT('# format=', FORMAT_ID), '$R$N');
				sBuffer := CONCAT(sBuffer, CONCAT(CONCAT('# sn=', sSN), '$R$N'));
				sBuffer := CONCAT(sBuffer, CONCAT(CONCAT('# start=', sStartIso), '$R$N'));
				sBuffer := CONCAT(sBuffer, CONCAT(CONCAT('# cycles_set=', UDINT_TO_STRING(nCyclesSet)), '$R$N'));
				sBuffer := CONCAT(sBuffer, CONCAT(CONCAT('# logged_cycle=', UDINT_TO_STRING(nCyclesSet)), '$R$N'));
				sBuffer := CONCAT(sBuffer, 't_ms,current,position_deg$R$N');
				nStep := 30;
			END_IF
			fbOpen(bExecute := FALSE);
		END_IF

	30, 50:	// write sBuffer: 30 = the header, 50 = one sample line
		sState := 'writing';
		fbWrite(sNetId := '', hFile := hFile, pWriteBuff := ADR(sBuffer), cbWriteLen := LEN(sBuffer),
			bExecute := TRUE, tTimeout := T#5S);
		IF NOT fbWrite.bBusy THEN
			IF fbWrite.bError THEN
				sLastError := CONCAT('write failed, run kept as ', sTmpPath);
				nErrors := nErrors + 1;
				bCompleted := FALSE;
				nStep := 60;
			ELSE
				nStep := 40;
			END_IF
			fbWrite(bExecute := FALSE);
		END_IF

	40:	// running: completion first - FB_Sequence ends a run with Step := 0 and bClose together
		sState := 'logging';
		IF bClose THEN
			bClose := FALSE;
			bAppend := FALSE;
			bCompleted := TRUE;
			nStep := 60;
		ELSIF bReset OR NOT bRunActive THEN
			sLastError := CONCAT('run stopped, kept as ', sTmpPath);
			bCompleted := FALSE;
			nStep := 60;
		ELSIF bAppend THEN
			bAppend := FALSE;
			sBuffer := CONCAT(UDINT_TO_STRING(nSamples * SAMPLE_MS), ',');
			sBuffer := CONCAT(sBuffer, CONCAT(REAL_TO_STRING(rCurrent), ','));
			sBuffer := CONCAT(sBuffer, CONCAT(DINT_TO_STRING(nPosition), '$R$N'));
			nSamples := nSamples + 1;
			nStep := 50;
		END_IF

	60:	// close; then rename if the run completed, else leave the .tmp
		sState := 'closing';
		fbClose(sNetId := '', hFile := hFile, bExecute := TRUE, tTimeout := T#5S);
		IF NOT fbClose.bBusy THEN
			IF fbClose.bError THEN
				sLastError := CONCAT('close failed: ', sTmpPath);
				nErrors := nErrors + 1;
				bCompleted := FALSE;
			END_IF
			bFileOpen := FALSE;
			fbClose(bExecute := FALSE);
			IF bCompleted THEN
				nStep := 70;
			ELSE
				nStep := 0;
			END_IF
		END_IF

	70:	// .tmp -> .log: from now on the run is visible to the report tool
		fbRename(sNetId := '', sOldName := sTmpPath, sNewName := sLogPath, ePath := PATH_GENERIC,
			bExecute := TRUE, tTimeout := T#5S);
		IF NOT fbRename.bBusy THEN
			IF fbRename.bError THEN
				sLastError := CONCAT('rename failed, run kept as ', sTmpPath);
				nErrors := nErrors + 1;
			ELSE
				sLastFile := sLogPath;
			END_IF
			fbRename(bExecute := FALSE);
			nStep := 0;
		END_IF
END_CASE

END_FUNCTION_BLOCK

// ---- RunLog/F_RunLogSnValid.TcPOU
// TRUE when sSN can go into a file name: 1..32 characters, each A-Z, a-z, 0-9 or '-'.
// The reader (elm-report) applies the same rule and rejects any other name.
FUNCTION F_RunLogSnValid : BOOL
VAR_INPUT
	sSN : STRING(32);
END_VAR
VAR
	i : INT;
	c : BYTE;
END_VAR

F_RunLogSnValid := LEN(sSN) >= 1;
FOR i := 0 TO LEN(sSN) - 1 DO
	c := sSN[i];
	IF NOT ((c >= 16#30 AND c <= 16#39)		// 0-9
		OR (c >= 16#41 AND c <= 16#5A)		// A-Z
		OR (c >= 16#61 AND c <= 16#7A)		// a-z
		OR c = 16#2D)						// -
	THEN
		F_RunLogSnValid := FALSE;
	END_IF
END_FOR

END_FUNCTION

// ---- POUs/OpenExplorer.TcPOU
PROGRAM OpenExplorer
VAR_INPUT
    NETID     : T_AmsNetId;
    PATHSTR   : T_MaxString;
    DIRNAME   : T_MaxString;
    COMNDLINE : T_MaxString;
    START     : BOOL;
    TMOUT     : TIME := DEFAULT_ADS_TIMEOUT;
	
	
	NT_StartProcess1      : NT_StartProcess;
NT_StartProcess_Busy  : BOOL;
NT_StartProcess_Err   : BOOL;
NT_StartProcess_ErrId : UDINT;
StartProcess          : BOOL;


END_VAR


NETID := '5.144.18.242.1.1';
PATHSTR := 'C:\WINNT\NOTEPAD.EXE';
DIRNAME := 'C:\WINNT';
COMNDLINE := 'win.ini';

NT_StartProcess1(
	NETID:= '5.144.18.242.1.1', 
	PATHSTR:= '\windows\explorer.exe', 
	DIRNAME:= '\windows' , 
	COMNDLINE:= 'explorer.exe' , 
	START:= gvl_io.OpenExplorer_cmd, 
	TMOUT:= TMOUT , 
	BUSY=> NT_StartProcess_Busy , 
	ERR=> NT_StartProcess_Err, 
	ERRID=> NT_StartProcess_ErrId);

END_PROGRAM

// ---- POUs/Sequence.TcPOU
PROGRAM Sequence
VAR
	Counter_1: CTU;
	temp: WORD;
	counter_PV: WORD;
	
	tempPosition, tempI:REAL;
	Position, Amper: INT;
	
	
	
	
	
END_VAR
VAR // added by the converter: edge detectors and wires of the graphical bodies
    _w1, _w2 : BOOL;
END_VAR

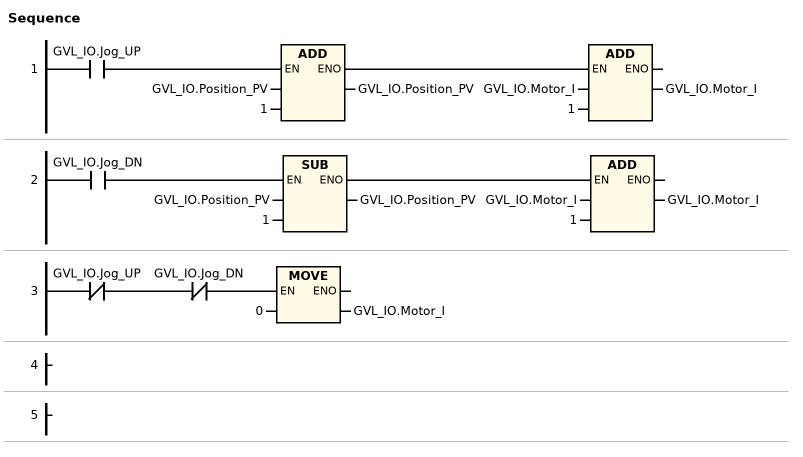
// NETWORK 1
_w1 := GVL_IO.Jog_UP;
IF _w1 THEN GVL_IO.Position_PV := GVL_IO.Position_PV + 1; END_IF
IF _w1 THEN GVL_IO.Motor_I := GVL_IO.Motor_I + 1; END_IF

// NETWORK 2
_w2 := GVL_IO.Jog_DN;
IF _w2 THEN GVL_IO.Position_PV := GVL_IO.Position_PV - 1; END_IF
IF _w2 THEN GVL_IO.Motor_I := GVL_IO.Motor_I + 1; END_IF

// NETWORK 3
IF NOT GVL_IO.Jog_UP AND NOT GVL_IO.Jog_DN THEN GVL_IO.Motor_I := 0; END_IF

// NETWORK 4

// NETWORK 5

END_PROGRAM

// ---- POUs/TestTorqueProfile.TcPOU
PROGRAM TestTorqueProfile
VAR
TorCmdMax : DINT := TRUNC( 3.0 * 1E6 / 10000);// TC*10e6/0x6076
MyTime : INT :=0;
tTimerValue     : LTIME ;//:= T#0S;
tTimeHr : UDINT;
END_VAR


//IF ServoCtrl.TargetTorque > TorCmdMax THEN
//	Ds402.DirUp := FALSE;
//END_IF
//
//IF ServoCtrl.TargetTorque < -TorCmdMax THEN
//	Ds402.DirUp := TRUE;
//END_IF
//		
//IF Ds402.DirUp THEN 
//	ServoCtrl.TargetTorque := ServoCtrl.TargetTorque+1;
//ELSE
//	ServoCtrl.TargetTorque := ServoCtrl.TargetTorque-1;
//END_IF

tTimerValue := LTIME();
tTimeHr := LTIME_TO_UDINT(tTimerValue) MOD  67108864 ;// 

MyTime := (MyTime +1) MOD  2048 ;
//for Ts=100usec: ServoCtrl.TargetTorque := TRUNC_INT( TorCmdMax * SIN(  tTimeHr * 6.28 *32.0 / 67108864.0 ));

// for Ts = 1ms
ServoCtrl.TargetTorque := TRUNC_INT( TorCmdMax * SIN(  tTimeHr * 6.28 *4.0 / 67108864.0 ));

// ServoCtrl.TargetTorque := TRUNC_INT( TorCmdMax * SIN(  MyTime * 6.28 * 25  / 2048.0 ));

END_PROGRAM

// ---- GlobalTextList.TcGTLO
TEXTLIST GlobalTextList
  787 = '\tPASSWORD'
  326 = '%.0d'
  626 = '%.0D'
  170 = '%.0d °'
  862 = '%.0D °'
  984 = '%.0f'
  839 = '%.0f °'
  138 = '%.0f °/s'
  923 = '%.1f'
  603 = '%.1f °'
  86 = '%0D °'
  846 = '%d'
  878 = '%d °'
  187 = '%D °'
  364 = '%s'
  511 = 'Accseleration A SP'
  411 = 'Accseleration B SP'
  200 = 'Accseleration slow SP'
  355 = 'Accseleration SP'
  856 = 'AL01Gripper Open Error'
  549 = 'AL02 Gripper Close Error'
  383 = 'AL02 Gripper close error'
  222 = 'AL02 Gripper Open Error'
  258 = 'AL03 Lock sensor error'
  151 = 'AL04 Homing error'
  101 = 'AL05 Motor error'
  209 = 'ALARMS'
  133 = 'AVR Current'
  424 = 'Brakes\nOPEN'
  301 = 'Cycle PV'
  612 = 'Cycle SP'
  142 = 'DN position\nSP'
  616 = 'DN position \nSP'
  772 = 'DN position SP'
  858 = 'EMERGENCY \nSTOP'
  938 = 'Emergency Stop'
  704 = 'Enable'
  654 = 'GO'
  296 = 'Gripper\nCLOSE'
  273 = 'Gripper\nOPEN'
  667 = 'Gripper Open Error'
  729 = 'Gripper open error'
  524 = 'HOMING'
  448 = 'JOG DN'
  530 = 'JOG UP'
  870 = 'Limit DN SP'
  867 = 'Limit UP SP'
  235 = 'MAX Current'
  997 = 'Motor\nDN'
  263 = 'Motor\nUP'
  985 = 'Motor I, Amper'
  94 = 'Motor slow\nDN'
  882 = 'Motor slow\nUP'
  217 = 'Please insert Shell\nAnd Approve'
  884 = 'Position DN A '
  17 = 'Position PV'
  582 = 'Position PV '
  983 = 'Position PV, mm'
  489 = 'Position SP'
  455 = 'Position UP A '
  927 = 'qx 0.0 \nclose gripper'
  551 = 'qx 0.0 \nopen gripper'
  891 = 'qx 0.0 \nstart motor'
  564 = 'R'
  745 = 'Reset'
  793 = 'SCV'
  864 = 'SETTINGS'
  147 = 'Settings'
  842 = 'Slow cycle'
  75 = 'SN'
  811 = 'Speed slow SP'
  831 = 'Speed SP'
  509 = 'START'
  556 = 'STOP'
  525 = 'UP position\nSP'
  885 = 'UP position SP'
  45 = 'V 1.0'
END_TEXTLIST

// ---- Screen/Alarm.TcVIS
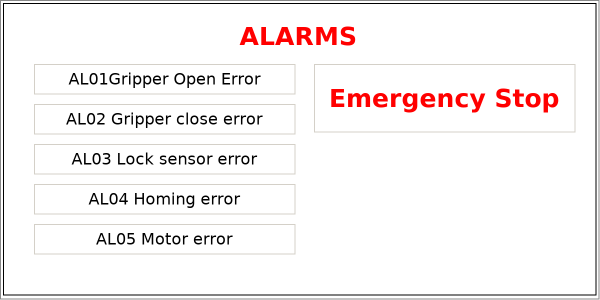
VISUALIZATION Alarm  // 600x300
    Rectangle (3,3 593x292)
    Label (217,21 163x30), "ALARMS"
    Textfield (34,64 261x30), "AL01Gripper Open Error", invisible if: GVL_IO.Gripper_Open_Error = 0
    Textfield (34,104 261x30), "AL02 Gripper close error", invisible if: GVL_IO.Gripper_Close_Error = 0
    Textfield (34,144 261x30), "AL03 Lock sensor error", invisible if: GVL_IO.SensorLock_Error = 0
    Textfield (34,184 261x30), "AL04 Homing error", invisible if: GVL_IO.Homing_Error = 0
    Textfield (34,224 261x30), "AL05 Motor error", invisible if: GVL_IO.Motor_Error = 0
    Textfield (314,64 261x68), "Emergency Stop", invisible if: GVL_IO.ixEmergancy_Stop
END_VISUALIZATION

// ---- Screen/Control_Panel.TcVIS
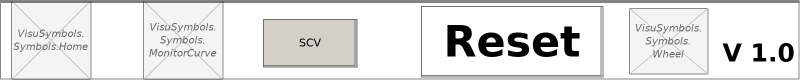
VISUALIZATION Control_Panel  // 800x80
    Image (11,0 80x80), image: VisuSymbols.Symbols.Home
        OnMouseClick: change screen: Overview_ATP
    Image (143,0 80x80), image: VisuSymbols.Symbols.MonitorCurve
        OnMouseClick: change screen: Graph
    Button (421,6 182x71), "Reset"
        tap GVL_IO.Reset
    Line (800,2) (0,2)
    Image (629,8 79x66), image: VisuSymbols.Symbols.Wheel
        OnMouseClick: change screen: Password
    Button (263,19 94x48), "SCV"
        tap GVL_IO.OpenExplorer_cmd
    Label (722,33 74x39), "V 1.0"
END_VISUALIZATION

// ---- Screen/Graph.TcVIS
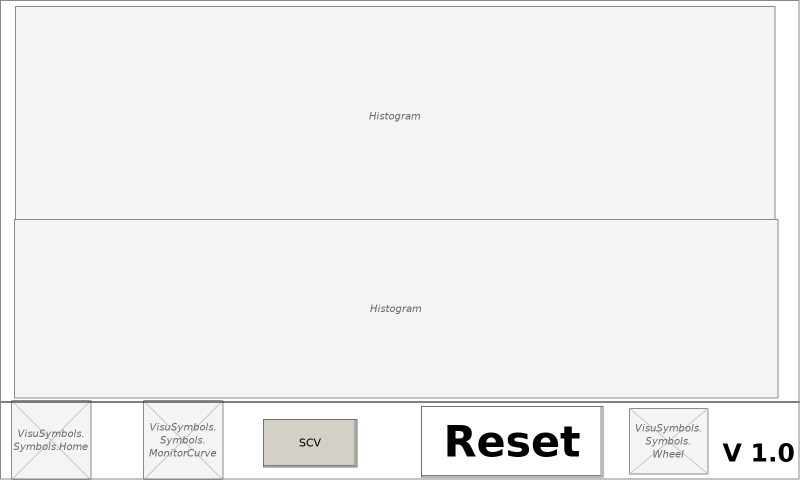
VISUALIZATION Graph  // 800x480
    Frame (0,400 800x80)
        shows Control_Panel()
    Histogram (15,6 760x220), scale format: %.0D, scale -500..500
        p518627256: Position PV, mm
        p1518820177: GVL_IO.Position_PV_mem
        p102497268: GVL_IO.Position_PV_mem
        p788070771: ARRAY [0..500] OF DINT
    Histogram (14,219 764x179), scale format: %.1f, scale 0..100
        p518627256: Motor I, Amper
        p1518820177: GVL_IO.Motor_I_mem
        p102497268: GVL_IO.Motor_I_mem
        p788070771: ARRAY [0..500] OF REAL
END_VISUALIZATION

// ---- Screen/Overview.TcVIS
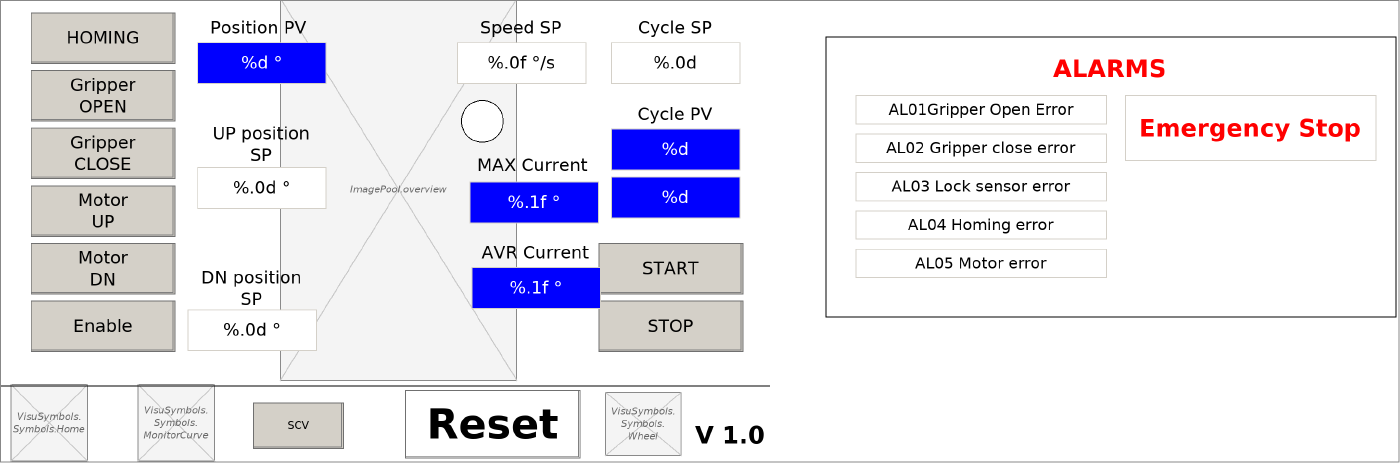
VISUALIZATION Overview  // 1455x482
    Button (32,13 150x53), "HOMING", colour toggle: GVL_IO.Homing_OK
        tap GVL_IO.Homing
    Button (32,73 150x53), "Gripper OPEN", colour toggle: GVL_IO.ixGripper_Unlock
        tap GVL_IO.Gripper_Open_cmd
    Button (32,133 150x53), "Gripper CLOSE", colour toggle: GVL_IO.TwoSensorLock
        tap GVL_IO.Gripper_Close_cmd
    Button (32,193 150x53), "Motor UP", colour toggle: GVL_IO.Motor_UP
        tap GVL_IO.Motor_UP
    Button (32,253 150x53), "Motor DN", colour toggle: GVL_IO.Motor_DN
        tap GVL_IO.Motor_DN
    Button (32,313 150x53), "Enable", colour toggle: GVL_IO.qxSTO_toDrive
        OnMouseClick: toggle GVL_IO.Enable_motor_cmd
    Frame (0,400 800x80)
        shows Control_Panel()
    Image (291,-2 246x398), image: ImagePool.overview
    Textfield (205,44 134x43), "%d °", text variable: GVL_IO.Position_PV_HMI
    Label (206,13 131x32), "Position PV"
    Label (206,125 131x50), "UP position SP"
    Textfield (205,174 134x43), "%.0d °", text variable: GVL_IO.Position_UP_SP
        OnMouseClick: write the text variable via Default
    Label (196,275 131x50), "DN position SP"
    Textfield (195,322 134x43), "%.0d °", text variable: GVL_IO.Position_DN_SP
        OnMouseClick: write the text variable via Default
    Label (636,13 131x32), "Cycle SP"
    Textfield (635,44 134x43), "%.0d", text variable: GVL_IO.Cycle_SP
        OnMouseClick: write the text variable via Default
    Textfield (475,44 134x43), "%.0f °/s", text variable: GVL_IO.Speed_SP
        OnMouseClick: write the text variable via Default
    Label (476,13 131x32), "Speed SP"
    Label (636,103 131x32), "Cycle PV"
    Textfield (635,134 134x43), "%d", text variable: GVL_IO.Cycle_PV
    Button (622,253 150x53), "START"
        tap GVL_IO.Start
    Button (622,313 150x53), "STOP", colour toggle: GVL_IO.Stop
        tap GVL_IO.Stop
    Textfield (635,184 134x43), "%d", text variable: ServoCtrl.Position
    Ellipse (479,104 44x44), colour toggle: GVL_IO.ixHome_Position
    Label (488,156 131x32), "MAX Current"
    Textfield (488,189 134x43), "%.1f °", text variable: GVL_IO.Motor_I_MAX
    Label (491,247 131x32), "AVR Current"
    Textfield (490,278 134x43), "%.1f °", text variable: GVL_IO.Motor_I_AVR
    Frame (855,35 600x300), invisible if: GVL_IO.Error = 0
        shows Alarm()
        p3560616238: -750
END_VISUALIZATION

// ---- Screen/Overview_ATP.TcVIS
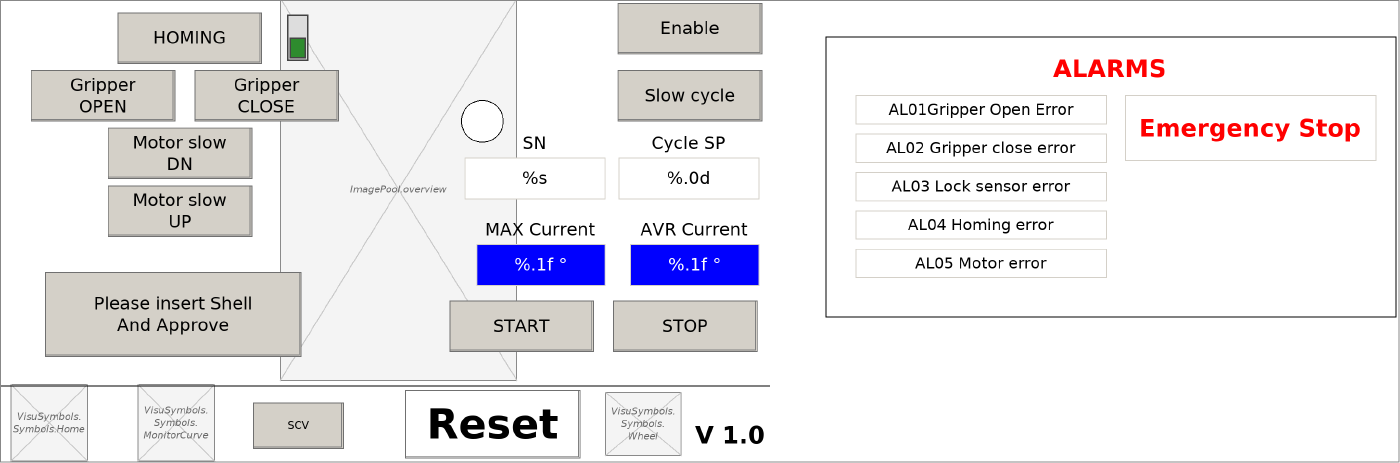
VISUALIZATION Overview_ATP  // 1455x482
    Button (122,13 150x53), "HOMING", colour toggle: GVL_IO.Homing_OK
        tap GVL_IO.Homing
    Button (32,73 150x53), "Gripper OPEN", colour toggle: GVL_IO.test_Gripper_open_OK, invisible if: not GVL_IO.Homing_OK
        tap GVL_IO.Gripper_Open_cmd
    Button (112,193 150x53), "Motor slow UP", colour toggle: GVL_IO.test_motor_slUP_ok, invisible if: not GVL_IO.Homing_OK
        tap GVL_IO.Motor_UP_slow_cmd
    Button (112,133 150x53), "Motor slow DN", colour toggle: GVL_IO.test_motor_sldown_ok, invisible if: not GVL_IO.Homing_OK
        tap GVL_IO.Motor_DN_slow_cmd
    Frame (0,400 800x80)
        shows Control_Panel()
    Image (291,-2 246x398), image: ImagePool.overview
    Label (206,13 131x32)
    Button (467,313 150x53), "START", invisible if: not GVL_IO.Homing_OK
        tap GVL_IO.ATP_start_cmd
    Button (637,313 150x53), "STOP", colour toggle: GVL_IO.Stop
        tap GVL_IO.Stop
    Ellipse (479,104 44x44), colour toggle: GVL_IO.ixHome_Position
    Button (202,73 150x53), "Gripper CLOSE", colour toggle: GVL_IO.test_Gripper_close_OK, invisible if: not GVL_IO.Homing_OK
        tap GVL_IO.Gripper_Close_cmd
    Button (642,3 150x53), "Enable", colour toggle: GVL_IO.qxSTO_toDrive
        OnMouseClick: toggle GVL_IO.Enable_motor_cmd
    Button (47,283 266x88), "Please insert Shell And Approve", colour toggle: GVL_IO.test_Insert_OK, invisible if: not GVL_IO.Homing_OK
        toggle GVL_IO.test_Insert_OK
    Button (642,73 150x53), "Slow cycle", colour toggle: GVL_IO.test_slowCycle_OK, invisible if: not GVL_IO.Homing_OK
        tap GVL_IO.Slow_cycle_cmd
    Label (644,133 143x32), "Cycle SP", invisible if: not GVL_IO.Homing_OK
    Textfield (643,164 146x43), "%.0d", text variable: GVL_IO.Cycle_SP, invisible if: not GVL_IO.Homing_OK
        OnMouseClick: write the text variable via Default
    Label (496,223 131x32), "MAX Current"
    Textfield (495,254 134x43), "%.1f °", text variable: GVL_IO.Motor_I_MAX
    Label (656,223 131x32), "AVR Current"
    Textfield (655,254 134x43), "%.1f °", text variable: GVL_IO.Motor_I_AVR
    DipSwitch (283,15 53x48), variable: GVL_IO.Homing_OK, behaviour: TOGGLE, style: Switch-DipSwitch-Green
    Frame (855,35 600x300), invisible if: GVL_IO.Error = 0
        shows Alarm()
        p3560616238: -750
    Label (484,133 143x32), "SN", invisible if: not GVL_IO.Homing_OK
    Textfield (483,164 146x43), "%s", text variable: GVL_RunLog.SN, invisible if: not GVL_IO.Homing_OK
        OnMouseClick: write the text variable via Default
END_VISUALIZATION

// ---- Screen/Servo.TcVIS
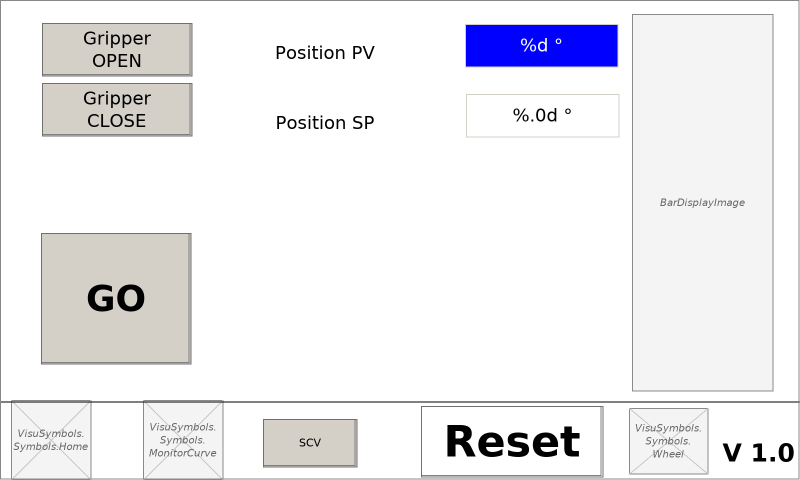
VISUALIZATION Servo  // 800x480
    Frame (0,400 800x80)
        shows Control_Panel()
    BarDisplayImage (632,14 141x377), value: ServoCtrl.ActualCurrent, style: BarDisplayImage-Gray, scale format: %.0d, scale 0..2000
        p518627256: Motor I, Amper
    Textfield (466,94 153x43), "%.0d °", text variable: GVL_IO.Position_SP
        OnMouseClick: write the text variable via Default
    Button (41,233 150x131), "GO"
        tap GVL_IO.GO_TO_cmd
    Label (250,38 150x30), "Position PV"
    Label (250,108 150x30), "Position SP"
    Textfield (465,24 153x43), "%d °", text variable: GVL_IO.Position_PV_HMI
    Button (42,23 150x53), "Gripper OPEN", colour toggle: GVL_IO.ixGripper_Unlock
        tap GVL_IO.Gripper_Open_cmd
    Button (42,83 150x53), "Gripper CLOSE", colour toggle: GVL_IO.TwoSensorLock
        tap GVL_IO.Gripper_Close_cmd
END_VISUALIZATION

// ---- Screen/Settings.TcVIS
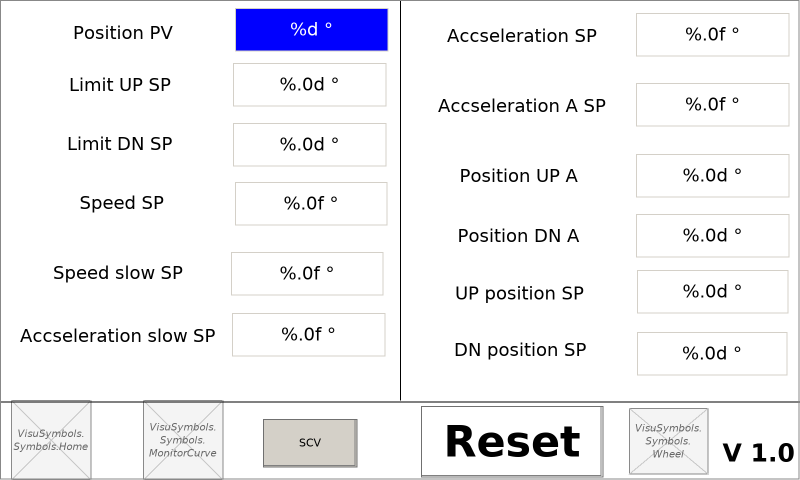
VISUALIZATION Settings  // 800x480
    Frame (0,400 800x80)
        shows Control_Panel()
    Textfield (636,154 153x43), "%.0d °", text variable: GVL_IO.Position_UP_A_SP
        OnMouseClick: write the text variable via Default
    Textfield (235,182 152x43), "%.0f °", text variable: GVL_IO.Speed_SP
        OnMouseClick: write the text variable via Default
    Label (20,18 206x30), "Position PV"
    Label (420,161 203x30), "Position UP A"
    Label (20,188 204x30), "Speed SP"
    Label (420,21 204x30), "Accseleration SP"
    Textfield (636,13 153x43), "%.0f °", text variable: GVL_IO.Accseleration_SP
        OnMouseClick: write the text variable via Default
    Textfield (235,8 153x43), "%d °", text variable: GVL_IO.Position_PV_HMI
    Label (17,70 206x30), "Limit UP SP"
    Textfield (233,63 153x43), "%.0d °", text variable: GVL_IO.Motor_Limit_UP
        OnMouseClick: write the text variable via Default
    Label (17,129 206x30), "Limit DN SP"
    Textfield (233,123 153x43), "%.0d °", text variable: GVL_IO.Motor_Limit_DN
        OnMouseClick: write the text variable via Default
    Line (400,0) (400,400)
    Label (420,221 203x30), "Position DN A"
    Textfield (636,214 153x43), "%.0d °", text variable: GVL_IO.Position_DN_A_SP
        OnMouseClick: write the text variable via Default
    Label (420,91 204x30), "Accseleration A SP"
    Textfield (636,83 153x43), "%.0f °", text variable: GVL_IO.Accseleration_A_SP
        OnMouseClick: write the text variable via Default
    Label (16,258 204x30), "Speed slow SP"
    Textfield (231,252 152x43), "%.0f °", text variable: GVL_IO.Speed_SP_slow
        OnMouseClick: write the text variable via Default
    Label (16,321 204x30), "Accseleration slow SP"
    Textfield (232,313 153x43), "%.0f °", text variable: GVL_IO.Accseleration_SP_slow
        OnMouseClick: write the text variable via Default
    Label (418,273 203x41), "UP position SP"
    Textfield (637,270 151x43), "%.0d °", text variable: GVL_IO.Position_UP_SP
        OnMouseClick: write the text variable via Default
    Label (403,325 235x50), "DN position SP"
    Textfield (637,332 150x43), "%.0d °", text variable: GVL_IO.Position_DN_SP
        OnMouseClick: write the text variable via Default
END_VISUALIZATION

// ---- Screen/Password.TcVIS
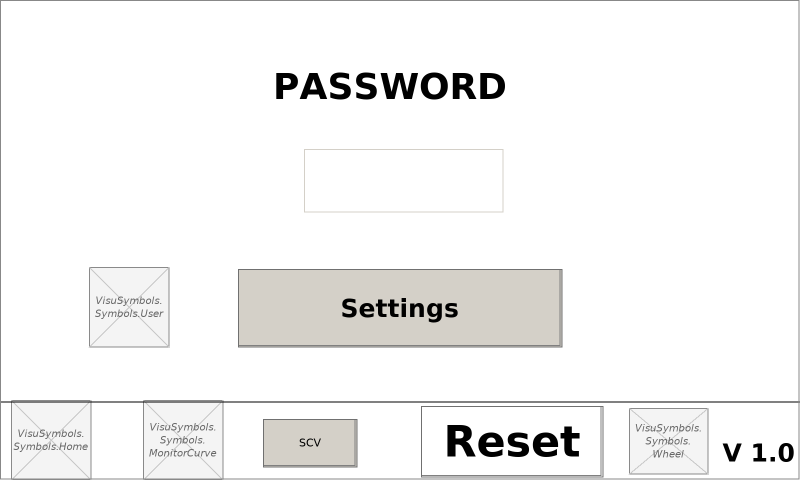
VISUALIZATION Password  // 800x480
    Frame (0,400 800x80)
        shows Control_Panel()
    Label (233,35 289x103), "PASSWORD"
    Textfield (304,149 199x63), text variable: GVL_IO.Password_IN
        OnMouseClick: write the text variable via Default, password
    Button (238,269 324x78), "Settings", invisible if: GVL_IO.Password_IN <> 9118
        OnMouseClick: change screen: Settings
    Image (89,267 80x80), invisible if: GVL_IO.Password_IN <> 9118, image: VisuSymbols.Symbols.User
        OnMouseClick: change screen: Overview
END_VISUALIZATION

// ---- VISUs/Visualization.TcVIS
VISUALIZATION Visualization  // 2x2
END_VISUALIZATION
